  MoveL 8876 to (499.7, 501.14, 17.4) mm, rotated rx 0 ry 90 rz 0 deg; joints [-12.119, -28.128, 111.655, -16.143, -82.918, 51.024]
  Set speed (120.0 mm/s)
  MoveL 8877 to (499.36, 500.49, 17.4) mm, rotated rx 0 ry 90 rz 0 deg; joints [-12.066, -28.137, 111.711, -16.087, -82.962, 51.005]
  Set speed (15.0 mm/s)
  Call Extruder(0.050)
  MoveL 8878 to (500.58, 499.27, 17.4) mm, rotated rx 0 ry 90 rz 0 deg; joints [-11.93, -28.118, 111.596, -15.954, -82.865, 51.017]
  Set speed (120.0 mm/s)
  MoveL 8879 to (500.25, 498.61, 17.4) mm, rotated rx 0 ry 90 rz 0 deg; joints [-11.876, -28.127, 111.653, -15.898, -82.909, 50.998]
  Set speed (15.0 mm/s)
  MoveL 8880 to (499.03, 499.83, 17.4) mm, rotated rx 0 ry 90 rz 0 deg; joints [-12.012, -28.145, 111.768, -16.032, -83.006, 50.986]
  Set speed (120.0 mm/s)
  MoveL 8881 to (498.69, 499.17, 17.4) mm, rotated rx 0 ry 90 rz 0 deg; joints [-11.958, -28.154, 111.824, -15.976, -83.05, 50.967]
  Set speed (15.0 mm/s)
  Call Extruder(0.050)
  MoveL 8882 to (499.91, 497.96, 17.4) mm, rotated rx 0 ry 90 rz 0 deg; joints [-11.823, -28.136, 111.709, -15.843, -82.953, 50.979]
  Set speed (120.0 mm/s)
  MoveL 8883 to (499.58, 497.3, 17.4) mm, rotated rx 0 ry 90 rz 0 deg; joints [-11.769, -28.145, 111.766, -15.787, -82.997, 50.96]
  Set speed (15.0 mm/s)
  MoveL 8884 to (498.36, 498.52, 17.4) mm, rotated rx 0 ry 90 rz 0 deg; joints [-11.905, -28.163, 111.881, -15.92, -83.094, 50.948]
  Set speed (120.0 mm/s)
  MoveL 8885 to (498.02, 497.86, 17.4) mm, rotated rx 0 ry 90 rz 0 deg; joints [-11.851, -28.172, 111.937, -15.864, -83.138, 50.929]
  Set speed (15.0 mm/s)
  Call Extruder(0.050)
  MoveL 8886 to (499.24, 496.65, 17.4) mm, rotated rx 0 ry 90 rz 0 deg; joints [-11.715, -28.154, 111.822, -15.731, -83.041, 50.942]
  Set speed (120.0 mm/s)
  MoveL 8887 to (498.91, 495.99, 17.4) mm, rotated rx 0 ry 90 rz 0 deg; joints [-11.662, -28.163, 111.878, -15.676, -83.085, 50.923]
  Set speed (15.0 mm/s)
  Call Extruder(0.050)
  MoveL 8888 to (497.69, 497.21, 17.4) mm, rotated rx 0 ry 90 rz 0 deg; joints [-11.797, -28.181, 111.993, -15.809, -83.183, 50.911]
  Set speed (120.0 mm/s)
  MoveL 8889 to (497.36, 496.55, 17.4) mm, rotated rx 0 ry 90 rz 0 deg; joints [-11.743, -28.189, 112.049, -15.753, -83.227, 50.892]
  Set speed (15.0 mm/s)
  Call Extruder(0.107)
  MoveL 8890 to (499.95, 493.96, 17.4) mm, rotated rx 0 ry 90 rz 0 deg; joints [-11.455, -28.151, 111.804, -15.47, -83.018, 50.918]
  Set speed (120.0 mm/s)
  MoveL 8891 to (498.96, 493.96, 17.4) mm, rotated rx 0 ry 90 rz 0 deg; joints [-11.474, -28.17, 111.922, -15.485, -83.115, 50.893]
  Set speed (15.0 mm/s)
  Call Extruder(0.080)
  MoveL 8892 to (497.02, 495.9, 17.4) mm, rotated rx 0 ry 90 rz 0 deg; joints [-11.689, -28.198, 112.105, -15.697, -83.271, 50.874]
  Set speed (120.0 mm/s)
  MoveL 8893 to (496.69, 495.24, 17.4) mm, rotated rx 0 ry 90 rz 0 deg; joints [-11.635, -28.206, 112.161, -15.641, -83.315, 50.855]
  Set speed (15.0 mm/s)
  Call Extruder(0.053)
  MoveL 8894 to (497.97, 493.96, 17.4) mm, rotated rx 0 ry 90 rz 0 deg; joints [-11.492, -28.188, 112.04, -15.501, -83.212, 50.868]
  Set speed (120.0 mm/s)
  MoveL 8895 to (496.98, 493.96, 17.4) mm, rotated rx 0 ry 90 rz 0 deg; joints [-11.511, -28.206, 112.158, -15.516, -83.309, 50.843]
  Set speed (15.0 mm/s)
  Call Extruder(0.026)
  MoveL 8896 to (496.35, 494.59, 17.4) mm, rotated rx 0 ry 90 rz 0 deg; joints [-11.58, -28.215, 112.217, -15.585, -83.359, 50.837]
  Set speed (120.0 mm/s)
  MoveL 8897 to (499.33, 495.57, 17.4) mm, rotated rx 0 ry 90 rz 0 deg; joints [-11.614, -28.156, 111.838, -15.629, -83.051, 50.927]
  Set speed (15.0 mm/s)
  Call Extruder(0.066)
  MoveL 8898 to (500.94, 493.96, 17.4) mm, rotated rx 0 ry 90 rz 0 deg; joints [-11.437, -28.132, 111.685, -15.455, -82.922, 50.943]
  Set speed (120.0 mm/s)
  MoveL 8899 to (501.93, 493.96, 17.4) mm, rotated rx 0 ry 90 rz 0 deg; joints [-11.418, -28.114, 111.567, -15.44, -82.825, 50.968]
  Set speed (15.0 mm/s)
  MoveL 8900 to (500.32, 495.57, 17.4) mm, rotated rx 0 ry 90 rz 0 deg; joints [-11.596, -28.138, 111.719, -15.614, -82.954, 50.952]
  Set speed (120.0 mm/s)
  MoveL 8901 to (501.31, 495.57, 17.4) mm, rotated rx 0 ry 90 rz 0 deg; joints [-11.577, -28.119, 111.601, -15.598, -82.858, 50.977]
  Set speed (15.0 mm/s)
  MoveL 8902 to (502.92, 493.96, 17.4) mm, rotated rx 0 ry 90 rz 0 deg; joints [-11.4, -28.095, 111.448, -15.425, -82.728, 50.992]
  Set speed (120.0 mm/s)
  MoveL 8903 to (503.91, 493.96, 17.4) mm, rotated rx 0 ry 90 rz 0 deg; joints [-11.382, -28.076, 111.329, -15.41, -82.632, 51.017]
  Set speed (15.0 mm/s)
  MoveL 8904 to (502.3, 495.57, 17.4) mm, rotated rx 0 ry 90 rz 0 deg; joints [-11.558, -28.1, 111.483, -15.583, -82.761, 51.002]
  Set speed (120.0 mm/s)
  MoveL 8905 to (503.29, 495.56, 17.4) mm, rotated rx 0 ry 90 rz 0 deg; joints [-11.54, -28.081, 111.364, -15.568, -82.665, 51.027]
  Set speed (15.0 mm/s)
  Call Extruder(0.035)
  MoveL 8906 to (504.15, 494.7, 17.4) mm, rotated rx 0 ry 90 rz 0 deg; joints [-11.445, -28.068, 111.281, -15.475, -82.595, 51.035]
  Set speed (120.0 mm/s)
  MoveL 8907 to (502.26, 502.54, 17.4) mm, rotated rx 0 ry 90 rz 0 deg; joints [-12.196, -28.073, 111.312, -16.231, -82.644, 51.114]
  Set speed (15.0 mm/s)
  Call Extruder(0.050)
  MoveL 8908 to (501.03, 503.76, 17.4) mm, rotated rx 0 ry 90 rz 0 deg; joints [-12.332, -28.091, 111.427, -16.364, -82.741, 51.102]
  MoveL 8909 to (500.91, 503.89, 17.4) mm, rotated rx 0 ry 90 rz 0 deg; joints [-12.346, -28.093, 111.438, -16.378, -82.751, 51.101]
  Set speed (120.0 mm/s)
  MoveL 8910 to (490.68, 490.68, 17.4) mm, rotated rx 0 ry 90 rz 0 deg; joints [-11.324, -28.329, 112.985, -15.308, -83.983, 50.637]
  Set speed (1000.0 mm/s)
  MoveL 8911 to (490.68, 490.68, 17.5) mm, rotated rx 0 ry 90 rz 0 deg; joints [-11.324, -28.339, 112.99, -15.308, -83.977, 50.638]
  Set speed (30.0 mm/s)
  Call Extruder(0.287)
  MoveL 8912 to (497.65, 497.65, 17.5) mm, rotated rx 0 ry 90 rz 0 deg; joints [-11.838, -28.19, 111.992, -15.851, -83.173, 50.918]
  MoveL 8913 to (497.78, 497.78, 17.5) mm, rotated rx 0 ry 90 rz 0 deg; joints [-11.847, -28.187, 111.974, -15.86, -83.159, 50.923]
  Set speed (120.0 mm/s)
  MoveL 8914 to (499.24, 500.76, 17.5) mm, rotated rx 0 ry 90 rz 0 deg; joints [-12.093, -28.148, 111.724, -16.115, -82.964, 51.008]
  Set speed (30.0 mm/s)
  Call Extruder(0.352)
  MoveL 8915 to (490.68, 509.32, 17.5) mm, rotated rx 0 ry 90 rz 0 deg; joints [-13.056, -28.269, 112.514, -17.061, -83.634, 50.914]
  MoveL 8916 to (490.56, 509.44, 17.5) mm, rotated rx 0 ry 90 rz 0 deg; joints [-13.07, -28.271, 112.525, -17.075, -83.643, 50.913]
  Set speed (120.0 mm/s)
  MoveL 8917 to (496.13, 506.03, 17.5) mm, rotated rx 0 ry 90 rz 0 deg; joints [-12.639, -28.185, 111.957, -16.657, -83.169, 51.01]
  Set speed (30.0 mm/s)
  Call Extruder(0.224)
  MoveL 8918 to (490.68, 500.58, 17.5) mm, rotated rx 0 ry 90 rz 0 deg; joints [-12.247, -28.304, 112.746, -16.241, -83.8, 50.78]
  Set speed (120.0 mm/s)
  MoveL 8919 to (490.68, 499.42, 17.5) mm, rotated rx 0 ry 90 rz 0 deg; joints [-12.139, -28.308, 112.775, -16.132, -83.821, 50.763]
  Set speed (30.0 mm/s)
  Call Extruder(0.215)
  MoveL 8920 to (495.89, 494.21, 17.5) mm, rotated rx 0 ry 90 rz 0 deg; joints [-11.554, -28.235, 112.286, -15.557, -83.405, 50.821]
  Set speed (120.0 mm/s)
  MoveL 8921 to (496.37, 493.73, 17.5) mm, rotated rx 0 ry 90 rz 0 deg; joints [-11.5, -28.228, 112.241, -15.504, -83.367, 50.826]
  Set speed (30.0 mm/s)
  Call Extruder(0.125)
  MoveL 8922 to (499.42, 490.68, 17.5) mm, rotated rx 0 ry 90 rz 0 deg; joints [-11.163, -28.184, 111.95, -15.172, -83.12, 50.857]
  Set speed (120.0 mm/s)
  MoveL 8923 to (500.58, 490.68, 17.5) mm, rotated rx 0 ry 90 rz 0 deg; joints [-11.141, -28.162, 111.812, -15.154, -83.006, 50.885]
  Set speed (30.0 mm/s)
  MoveL 8924 to (503.63, 493.73, 17.5) mm, rotated rx 0 ry 90 rz 0 deg; joints [-11.366, -28.092, 111.374, -15.392, -82.658, 51.008]
  Set speed (120.0 mm/s)
  MoveL 8925 to (504.39, 494.49, 17.5) mm, rotated rx 0 ry 90 rz 0 deg; joints [-11.421, -28.075, 111.263, -15.451, -82.57, 51.039]
  Set speed (30.0 mm/s)
  Call Extruder(0.203)
  MoveL 8926 to (509.32, 499.42, 17.5) mm, rotated rx 0 ry 90 rz 0 deg; joints [-11.777, -27.956, 110.548, -15.832, -82.008, 51.244]
  Set speed (120.0 mm/s)
  MoveL 8927 to (509.32, 500.58, 17.5) mm, rotated rx 0 ry 90 rz 0 deg; joints [-11.882, -27.951, 110.519, -15.939, -81.988, 51.264]
  Set speed (30.0 mm/s)
  Call Extruder(0.212)
  MoveL 8928 to (504.16, 505.74, 17.5) mm, rotated rx 0 ry 90 rz 0 deg; joints [-12.449, -28.032, 111.006, -16.495, -82.397, 51.219]
  Set speed (120.0 mm/s)
  MoveL 8929 to (503.3, 506.6, 17.5) mm, rotated rx 0 ry 90 rz 0 deg; joints [-12.544, -28.046, 111.086, -16.589, -82.465, 51.211]
  Set speed (30.0 mm/s)
  Call Extruder(0.112)
  MoveL 8930 to (500.58, 509.32, 17.5) mm, rotated rx 0 ry 90 rz 0 deg; joints [-12.847, -28.087, 111.338, -16.886, -82.677, 51.184]
  Set speed (120.0 mm/s)
  MoveL 8931 to (499.42, 509.32, 17.5) mm, rotated rx 0 ry 90 rz 0 deg; joints [-12.872, -28.109, 111.476, -16.906, -82.789, 51.153]
  Set speed (30.0 mm/s)
  Call Extruder(0.112)
  MoveL 8932 to (496.7, 506.6, 17.5) mm, rotated rx 0 ry 90 rz 0 deg; joints [-12.679, -28.172, 111.874, -16.701, -83.103, 51.035]
  MoveL 8933 to (496.57, 506.47, 17.5) mm, rotated rx 0 ry 90 rz 0 deg; joints [-12.67, -28.175, 111.892, -16.691, -83.118, 51.029]
  Set speed (120.0 mm/s)
  MoveL 8934 to (502.51, 502.51, 17.5) mm, rotated rx 0 ry 90 rz 0 deg; joints [-12.188, -28.079, 111.289, -16.224, -82.615, 51.121]
  Set speed (30.0 mm/s)
  Call Extruder(0.280)
  MoveL 8935 to (509.32, 509.32, 17.5) mm, rotated rx 0 ry 90 rz 0 deg; joints [-12.669, -27.912, 110.29, -16.74, -81.835, 51.418]
  MoveL 8936 to (509.44, 509.44, 17.5) mm, rotated rx 0 ry 90 rz 0 deg; joints [-12.677, -27.908, 110.272, -16.75, -81.821, 51.423]
  Set speed (120.0 mm/s)
  MoveL 8937 to (500.81, 499.19, 17.5) mm, rotated rx 0 ry 90 rz 0 deg; joints [-11.919, -28.125, 111.576, -15.943, -82.839, 51.023]
  Set speed (30.0 mm/s)
  Call Extruder(0.140)
  MoveL 8938 to (504.2, 495.8, 17.5) mm, rotated rx 0 ry 90 rz 0 deg; joints [-11.544, -28.073, 111.255, -15.576, -82.567, 51.055]
  Set speed (120.0 mm/s)
  MoveL 8939 to (504.39, 495.61, 17.5) mm, rotated rx 0 ry 90 rz 0 deg; joints [-11.523, -28.07, 111.236, -15.555, -82.552, 51.057]
  Set speed (30.0 mm/s)
  Call Extruder(0.203)
  MoveL 8940 to (509.32, 490.68, 17.5) mm, rotated rx 0 ry 90 rz 0 deg; joints [-10.985, -27.992, 110.761, -15.026, -82.151, 51.098]
  MoveL 8941 to (509.44, 490.56, 17.5) mm, rotated rx 0 ry 90 rz 0 deg; joints [-10.972, -27.99, 110.749, -15.013, -82.141, 51.099]
  Set speed (120.0 mm/s)
  MoveL 8942 to (490.47, 509.53, 17.5) mm, rotated rx 0 ry 90 rz 0 deg; joints [-13.08, -28.272, 112.533, -17.085, -83.65, 50.912]
  Set speed (1000.0 mm/s)
  MoveL 8943 to (490.4, 509.6, 17.5) mm, rotated rx 0 ry 90 rz 0 deg; joints [-13.088, -28.273, 112.539, -17.093, -83.655, 50.911]
  Set speed (15.0 mm/s)
  Call Extruder(0.559)
  MoveL 8944 to (490.4, 490.4, 17.5) mm, rotated rx 0 ry 90 rz 0 deg; joints [-11.303, -28.345, 113.03, -15.286, -84.009, 50.628]
  MoveL 8945 to (509.6, 490.4, 17.5) mm, rotated rx 0 ry 90 rz 0 deg; joints [-10.955, -27.987, 110.733, -14.997, -82.128, 51.101]
  MoveL 8946 to (509.6, 509.6, 17.5) mm, rotated rx 0 ry 90 rz 0 deg; joints [-12.688, -27.904, 110.248, -16.761, -81.803, 51.43]
  MoveL 8947 to (490.4, 509.6, 17.5) mm, rotated rx 0 ry 90 rz 0 deg; joints [-13.088, -28.273, 112.539, -17.093, -83.655, 50.911]
  Set speed (120.0 mm/s)
  MoveL 8948 to (490.4, 509.2, 17.5) mm, rotated rx 0 ry 90 rz 0 deg; joints [-13.051, -28.275, 112.55, -17.055, -83.663, 50.905]
  Set speed (1000.0 mm/s)
  MoveL 8949 to (490.5, 509.2, 17.5) mm, rotated rx 0 ry 90 rz 0 deg; joints [-13.049, -28.273, 112.538, -17.054, -83.653, 50.908]
  Set speed (1000.0 mm/s)
  MoveL 8950 to (496.05, 506.68, 17.5) mm, rotated rx 0 ry 90 rz 0 deg; joints [-12.7, -28.184, 111.949, -16.719, -83.165, 51.018]
  Set speed (15.0 mm/s)
  Call Extruder(0.065)
  MoveL 8951 to (496.05, 504.44, 17.5) mm, rotated rx 0 ry 90 rz 0 deg; joints [-12.495, -28.193, 112.009, -16.511, -83.207, 50.983]
  Call Extruder(0.145)
  MoveL 8952 to (501.03, 504.44, 17.5) mm, rotated rx 0 ry 90 rz 0 deg; joints [-12.394, -28.099, 111.415, -16.428, -82.724, 51.115]
  Call Extruder(0.353)
  MoveL 8953 to (495.52, 493.65, 17.5) mm, rotated rx 0 ry 90 rz 0 deg; joints [-11.509, -28.244, 112.344, -15.51, -83.451, 50.803]
  Call Extruder(0.261)
  MoveL 8954 to (504.47, 493.65, 17.5) mm, rotated rx 0 ry 90 rz 0 deg; joints [-11.343, -28.076, 111.274, -15.372, -82.576, 51.027]
  Call Extruder(0.065)
  MoveL 8955 to (504.47, 495.88, 17.5) mm, rotated rx 0 ry 90 rz 0 deg; joints [-11.547, -28.068, 111.22, -15.579, -82.539, 51.063]
  Call Extruder(0.153)
  MoveL 8956 to (499.2, 495.88, 17.5) mm, rotated rx 0 ry 90 rz 0 deg; joints [-11.646, -28.168, 111.85, -15.661, -83.053, 50.93]
  Call Extruder(0.353)
  MoveL 8957 to (504.73, 506.68, 17.5) mm, rotated rx 0 ry 90 rz 0 deg; joints [-12.523, -28.017, 110.912, -16.573, -82.325, 51.25]
  Call Extruder(0.253)
  MoveL 8958 to (496.05, 506.68, 17.5) mm, rotated rx 0 ry 90 rz 0 deg; joints [-12.7, -28.184, 111.949, -16.719, -83.165, 51.018]
  Set speed (120.0 mm/s)
  MoveL 8959 to (496.46, 506.36, 17.5) mm, rotated rx 0 ry 90 rz 0 deg; joints [-12.662, -28.177, 111.908, -16.683, -83.131, 51.025]
  Set speed (15.0 mm/s)
  Call Extruder(0.004)
  MoveL 8960 to (496.36, 506.26, 17.5) mm, rotated rx 0 ry 90 rz 0 deg; joints [-12.655, -28.18, 111.923, -16.675, -83.142, 51.02]
  Set speed (120.0 mm/s)
  MoveL 8961 to (496.36, 505.27, 17.5) mm, rotated rx 0 ry 90 rz 0 deg; joints [-12.564, -28.184, 111.95, -16.583, -83.161, 51.004]
  Set speed (15.0 mm/s)
  Call Extruder(0.045)
  MoveL 8962 to (497.45, 506.36, 17.5) mm, rotated rx 0 ry 90 rz 0 deg; joints [-12.642, -28.159, 111.791, -16.666, -83.035, 51.051]
  Set speed (120.0 mm/s)
  MoveL 8963 to (498.44, 506.36, 17.5) mm, rotated rx 0 ry 90 rz 0 deg; joints [-12.622, -28.14, 111.673, -16.649, -82.939, 51.078]
  Set speed (15.0 mm/s)
  Call Extruder(0.066)
  MoveL 8964 to (496.84, 504.76, 17.5) mm, rotated rx 0 ry 90 rz 0 deg; joints [-12.508, -28.177, 111.906, -16.527, -83.124, 51.009]
  Set speed (120.0 mm/s)
  MoveL 8965 to (497.83, 504.76, 17.5) mm, rotated rx 0 ry 90 rz 0 deg; joints [-12.488, -28.158, 111.788, -16.51, -83.028, 51.035]
  Set speed (15.0 mm/s)
  MoveL 8966 to (499.43, 506.36, 17.5) mm, rotated rx 0 ry 90 rz 0 deg; joints [-12.602, -28.121, 111.555, -16.632, -82.843, 51.104]
  Set speed (120.0 mm/s)
  MoveL 8967 to (500.42, 506.36, 17.5) mm, rotated rx 0 ry 90 rz 0 deg; joints [-12.581, -28.103, 111.437, -16.615, -82.747, 51.13]
  Set speed (15.0 mm/s)
  MoveL 8968 to (498.82, 504.76, 17.5) mm, rotated rx 0 ry 90 rz 0 deg; joints [-12.468, -28.14, 111.67, -16.493, -82.932, 51.061]
  Set speed (120.0 mm/s)
  MoveL 8969 to (499.81, 504.76, 17.5) mm, rotated rx 0 ry 90 rz 0 deg; joints [-12.448, -28.121, 111.552, -16.477, -82.836, 51.088]
  Set speed (15.0 mm/s)
  MoveL 8970 to (501.41, 506.36, 17.5) mm, rotated rx 0 ry 90 rz 0 deg; joints [-12.561, -28.083, 111.318, -16.599, -82.652, 51.157]
  Set speed (120.0 mm/s)
  MoveL 8971 to (502.4, 506.36, 17.5) mm, rotated rx 0 ry 90 rz 0 deg; joints [-12.541, -28.064, 111.2, -16.582, -82.556, 51.183]
  Set speed (15.0 mm/s)
  MoveL 8972 to (500.8, 504.76, 17.5) mm, rotated rx 0 ry 90 rz 0 deg; joints [-12.428, -28.102, 111.434, -16.46, -82.74, 51.114]
  Set speed (120.0 mm/s)
  MoveL 8973 to (501.28, 504.25, 17.5) mm, rotated rx 0 ry 90 rz 0 deg; joints [-12.372, -28.095, 111.389, -16.406, -82.703, 51.118]
  Set speed (15.0 mm/s)
  Call Extruder(0.087)
  MoveL 8974 to (503.39, 506.36, 17.5) mm, rotated rx 0 ry 90 rz 0 deg; joints [-12.521, -28.045, 111.081, -16.566, -82.46, 51.209]
  Set speed (120.0 mm/s)
  MoveL 8975 to (504.04, 506.02, 17.5) mm, rotated rx 0 ry 90 rz 0 deg; joints [-12.477, -28.034, 111.013, -16.523, -82.404, 51.22]
  Set speed (15.0 mm/s)
  Call Extruder(0.156)
  MoveL 8976 to (500.25, 502.23, 17.5) mm, rotated rx 0 ry 90 rz 0 deg; joints [-12.208, -28.123, 111.565, -16.235, -82.839, 51.058]
  MoveL 8977 to (500.13, 502.11, 17.5) mm, rotated rx 0 ry 90 rz 0 deg; joints [-12.199, -28.126, 111.583, -16.226, -82.853, 51.053]
  Set speed (120.0 mm/s)
  MoveL 8978 to (501.96, 501.96, 17.5) mm, rotated rx 0 ry 90 rz 0 deg; joints [-12.15, -28.091, 111.367, -16.182, -82.678, 51.098]
  Set speed (15.0 mm/s)
  Call Extruder(0.155)
  MoveL 8979 to (498.19, 498.19, 17.5) mm, rotated rx 0 ry 90 rz 0 deg; joints [-11.878, -28.178, 111.914, -15.892, -83.111, 50.94]
  MoveL 8980 to (498.07, 498.07, 17.5) mm, rotated rx 0 ry 90 rz 0 deg; joints [-11.869, -28.181, 111.932, -15.883, -83.125, 50.935]
  Set speed (120.0 mm/s)
  MoveL 8981 to (499.89, 497.91, 17.5) mm, rotated rx 0 ry 90 rz 0 deg; joints [-11.819, -28.147, 111.718, -15.839, -82.951, 50.979]
  Set speed (15.0 mm/s)
  Call Extruder(0.155)
  MoveL 8982 to (496.13, 494.15, 17.5) mm, rotated rx 0 ry 90 rz 0 deg; joints [-11.544, -28.231, 112.26, -15.548, -83.383, 50.826]
  Set speed (120.0 mm/s)
  MoveL 8983 to (496.93, 493.96, 17.5) mm, rotated rx 0 ry 90 rz 0 deg; joints [-11.512, -28.217, 112.168, -15.517, -83.308, 50.844]
  Set speed (15.0 mm/s)
  Call Extruder(0.079)
  MoveL 8984 to (498.85, 495.88, 17.5) mm, rotated rx 0 ry 90 rz 0 deg; joints [-11.652, -28.175, 111.893, -15.666, -83.087, 50.921]
  Set speed (120.0 mm/s)
  MoveL 8985 to (499.52, 495.56, 17.5) mm, rotated rx 0 ry 90 rz 0 deg; joints [-11.611, -28.163, 111.82, -15.626, -83.027, 50.934]
  Set speed (15.0 mm/s)
  Call Extruder(0.066)
  MoveL 8986 to (497.92, 493.96, 17.5) mm, rotated rx 0 ry 90 rz 0 deg; joints [-11.493, -28.199, 112.051, -15.502, -83.211, 50.869]
  Set speed (120.0 mm/s)
  MoveL 8987 to (498.91, 493.96, 17.5) mm, rotated rx 0 ry 90 rz 0 deg; joints [-11.475, -28.181, 111.932, -15.486, -83.114, 50.894]
  Set speed (15.0 mm/s)
  MoveL 8988 to (500.51, 495.57, 17.5) mm, rotated rx 0 ry 90 rz 0 deg; joints [-11.592, -28.145, 111.702, -15.611, -82.93, 50.959]
  Set speed (120.0 mm/s)
  MoveL 8989 to (501.5, 495.56, 17.5) mm, rotated rx 0 ry 90 rz 0 deg; joints [-11.573, -28.126, 111.583, -15.595, -82.834, 50.984]
  Set speed (15.0 mm/s)
  MoveL 8990 to (499.9, 493.96, 17.5) mm, rotated rx 0 ry 90 rz 0 deg; joints [-11.456, -28.162, 111.814, -15.471, -83.018, 50.918]
  Set speed (120.0 mm/s)
  MoveL 8991 to (500.89, 493.96, 17.5) mm, rotated rx 0 ry 90 rz 0 deg; joints [-11.438, -28.144, 111.696, -15.456, -82.921, 50.943]
  Set speed (15.0 mm/s)
  MoveL 8992 to (502.49, 495.56, 17.5) mm, rotated rx 0 ry 90 rz 0 deg; joints [-11.555, -28.107, 111.465, -15.58, -82.737, 51.009]
  Set speed (120.0 mm/s)
  MoveL 8993 to (503.48, 495.56, 17.5) mm, rotated rx 0 ry 90 rz 0 deg; joints [-11.536, -28.088, 111.346, -15.565, -82.641, 51.033]
  Set speed (15.0 mm/s)
  MoveL 8994 to (501.88, 493.96, 17.5) mm, rotated rx 0 ry 90 rz 0 deg; joints [-11.419, -28.125, 111.577, -15.44, -82.824, 50.968]
  Set speed (120.0 mm/s)
  MoveL 8995 to (502.87, 493.96, 17.5) mm, rotated rx 0 ry 90 rz 0 deg; joints [-11.401, -28.106, 111.459, -15.425, -82.727, 50.993]
  Set speed (15.0 mm/s)
  Call Extruder(0.053)
  MoveL 8996 to (504.16, 495.25, 17.5) mm, rotated rx 0 ry 90 rz 0 deg; joints [-11.495, -28.076, 111.273, -15.525, -82.581, 51.045]
  Set speed (120.0 mm/s)
  MoveL 8997 to (504.16, 494.26, 17.5) mm, rotated rx 0 ry 90 rz 0 deg; joints [-11.404, -28.08, 111.297, -15.433, -82.597, 51.029]
  Set speed (15.0 mm/s)
  Call Extruder(0.012)
  MoveL 8998 to (503.86, 493.96, 17.5) mm, rotated rx 0 ry 90 rz 0 deg; joints [-11.383, -28.087, 111.34, -15.41, -82.631, 51.017]
  Set speed (120.0 mm/s)
  MoveL 8999 to (500.93, 499.94, 17.5) mm, rotated rx 0 ry 90 rz 0 deg; joints [-11.985, -28.12, 111.543, -16.011, -82.814, 51.038]
  Set speed (15.0 mm/s)
  Call Extruder(0.155)
  MoveL 9000 to (497.16, 496.17, 17.5) mm, rotated rx 0 ry 90 rz 0 deg; joints [-11.711, -28.205, 112.087, -15.72, -83.247, 50.883]
  MoveL 9001 to (497.04, 496.05, 17.5) mm, rotated rx 0 ry 90 rz 0 deg; joints [-11.702, -28.208, 112.105, -15.711, -83.261, 50.878]
  Set speed (120.0 mm/s)
  MoveL 9002 to (499.22, 500.21, 17.5) mm, rotated rx 0 ry 90 rz 0 deg; joints [-12.043, -28.151, 111.74, -16.064, -82.975, 50.999]
  Set speed (15.0 mm/s)
  Call Extruder(0.156)
  MoveL 9003 to (503, 503.99, 17.5) mm, rotated rx 0 ry 90 rz 0 deg; joints [-12.314, -28.063, 111.19, -16.353, -82.541, 51.159]
  MoveL 9004 to (503.13, 504.12, 17.5) mm, rotated rx 0 ry 90 rz 0 deg; joints [-12.323, -28.06, 111.173, -16.363, -82.527, 51.164]
  Set speed (120.0 mm/s)
  MoveL 9005 to (490.68, 490.68, 17.5) mm, rotated rx 0 ry 90 rz 0 deg; joints [-11.324, -28.339, 112.99, -15.308, -83.977, 50.638]
  Set speed (1000.0 mm/s)
  MoveL 9006 to (490.68, 490.68, 17.6) mm, rotated rx 0 ry 90 rz 0 deg; joints [-11.324, -28.35, 112.995, -15.308, -83.972, 50.64]
  Set speed (30.0 mm/s)
  Call Extruder(0.287)
  MoveL 9007 to (497.65, 497.65, 17.6) mm, rotated rx 0 ry 90 rz 0 deg; joints [-11.838, -28.201, 111.997, -15.851, -83.168, 50.92]
  MoveL 9008 to (497.78, 497.78, 17.6) mm, rotated rx 0 ry 90 rz 0 deg; joints [-11.847, -28.198, 111.979, -15.861, -83.154, 50.925]
  Set speed (120.0 mm/s)
  MoveL 9009 to (499.24, 500.76, 17.6) mm, rotated rx 0 ry 90 rz 0 deg; joints [-12.093, -28.159, 111.729, -16.115, -82.959, 51.009]
  Set speed (30.0 mm/s)
  Call Extruder(0.352)
  MoveL 9010 to (490.68, 509.32, 17.6) mm, rotated rx 0 ry 90 rz 0 deg; joints [-13.056, -28.28, 112.519, -17.062, -83.628, 50.916]
  MoveL 9011 to (490.56, 509.44, 17.6) mm, rotated rx 0 ry 90 rz 0 deg; joints [-13.07, -28.282, 112.53, -17.075, -83.638, 50.915]
  Set speed (120.0 mm/s)
  MoveL 9012 to (496.13, 506.03, 17.6) mm, rotated rx 0 ry 90 rz 0 deg; joints [-12.639, -28.195, 111.962, -16.658, -83.164, 51.012]
  Set speed (30.0 mm/s)
  Call Extruder(0.224)
  MoveL 9013 to (490.68, 500.58, 17.6) mm, rotated rx 0 ry 90 rz 0 deg; joints [-12.247, -28.314, 112.751, -16.242, -83.795, 50.782]
  Set speed (120.0 mm/s)
  MoveL 9014 to (490.68, 499.42, 17.6) mm, rotated rx 0 ry 90 rz 0 deg; joints [-12.139, -28.319, 112.78, -16.132, -83.816, 50.765]
  Set speed (30.0 mm/s)
  Call Extruder(0.215)
  MoveL 9015 to (495.89, 494.21, 17.6) mm, rotated rx 0 ry 90 rz 0 deg; joints [-11.554, -28.246, 112.291, -15.557, -83.4, 50.822]
  Set speed (120.0 mm/s)
  MoveL 9016 to (496.37, 493.73, 17.6) mm, rotated rx 0 ry 90 rz 0 deg; joints [-11.5, -28.239, 112.246, -15.504, -83.361, 50.827]
  Set speed (30.0 mm/s)
  Call Extruder(0.125)
  MoveL 9017 to (499.42, 490.68, 17.6) mm, rotated rx 0 ry 90 rz 0 deg; joints [-11.163, -28.194, 111.955, -15.172, -83.114, 50.858]
  Set speed (120.0 mm/s)
  MoveL 9018 to (500.58, 490.68, 17.6) mm, rotated rx 0 ry 90 rz 0 deg; joints [-11.141, -28.173, 111.817, -15.154, -83.001, 50.887]
  Set speed (30.0 mm/s)
  MoveL 9019 to (503.63, 493.73, 17.6) mm, rotated rx 0 ry 90 rz 0 deg; joints [-11.366, -28.103, 111.379, -15.392, -82.652, 51.009]
  Set speed (120.0 mm/s)
  MoveL 9020 to (504.39, 494.49, 17.6) mm, rotated rx 0 ry 90 rz 0 deg; joints [-11.421, -28.085, 111.268, -15.452, -82.565, 51.04]
  Set speed (30.0 mm/s)
  Call Extruder(0.203)
  MoveL 9021 to (509.32, 499.42, 17.6) mm, rotated rx 0 ry 90 rz 0 deg; joints [-11.777, -27.966, 110.553, -15.832, -82.003, 51.245]
  Set speed (120.0 mm/s)
  MoveL 9022 to (509.32, 500.58, 17.6) mm, rotated rx 0 ry 90 rz 0 deg; joints [-11.882, -27.961, 110.524, -15.939, -81.983, 51.265]
  Set speed (30.0 mm/s)
  Call Extruder(0.212)
  MoveL 9023 to (504.16, 505.74, 17.6) mm, rotated rx 0 ry 90 rz 0 deg; joints [-12.449, -28.043, 111.011, -16.496, -82.392, 51.22]
  Set speed (120.0 mm/s)
  MoveL 9024 to (503.3, 506.6, 17.6) mm, rotated rx 0 ry 90 rz 0 deg; joints [-12.544, -28.056, 111.091, -16.589, -82.46, 51.212]
  Set speed (30.0 mm/s)
  Call Extruder(0.112)
  MoveL 9025 to (500.58, 509.32, 17.6) mm, rotated rx 0 ry 90 rz 0 deg; joints [-12.847, -28.097, 111.343, -16.887, -82.672, 51.186]
  Set speed (120.0 mm/s)
  MoveL 9026 to (499.42, 509.32, 17.6) mm, rotated rx 0 ry 90 rz 0 deg; joints [-12.872, -28.12, 111.482, -16.906, -82.784, 51.155]
  Set speed (30.0 mm/s)
  Call Extruder(0.112)
  MoveL 9027 to (496.7, 506.6, 17.6) mm, rotated rx 0 ry 90 rz 0 deg; joints [-12.679, -28.182, 111.879, -16.701, -83.098, 51.036]
  MoveL 9028 to (496.57, 506.47, 17.6) mm, rotated rx 0 ry 90 rz 0 deg; joints [-12.67, -28.185, 111.897, -16.691, -83.112, 51.031]
  Set speed (120.0 mm/s)
  MoveL 9029 to (502.51, 502.51, 17.6) mm, rotated rx 0 ry 90 rz 0 deg; joints [-12.188, -28.089, 111.294, -16.224, -82.61, 51.123]
  Set speed (30.0 mm/s)
  Call Extruder(0.280)
  MoveL 9030 to (509.32, 509.32, 17.6) mm, rotated rx 0 ry 90 rz 0 deg; joints [-12.669, -27.922, 110.295, -16.741, -81.83, 51.419]
  MoveL 9031 to (509.44, 509.44, 17.6) mm, rotated rx 0 ry 90 rz 0 deg; joints [-12.677, -27.919, 110.277, -16.75, -81.816, 51.425]
  Set speed (120.0 mm/s)
  MoveL 9032 to (500.81, 499.19, 17.6) mm, rotated rx 0 ry 90 rz 0 deg; joints [-11.919, -28.135, 111.581, -15.944, -82.834, 51.025]
  Set speed (30.0 mm/s)
  Call Extruder(0.140)
  MoveL 9033 to (504.2, 495.8, 17.6) mm, rotated rx 0 ry 90 rz 0 deg; joints [-11.544, -28.084, 111.26, -15.576, -82.562, 51.057]
  Set speed (120.0 mm/s)
  MoveL 9034 to (504.39, 495.61, 17.6) mm, rotated rx 0 ry 90 rz 0 deg; joints [-11.523, -28.081, 111.241, -15.555, -82.546, 51.058]
  Set speed (30.0 mm/s)
  Call Extruder(0.203)
  MoveL 9035 to (509.32, 490.68, 17.6) mm, rotated rx 0 ry 90 rz 0 deg; joints [-10.985, -28.002, 110.766, -15.027, -82.146, 51.1]
  MoveL 9036 to (509.44, 490.56, 17.6) mm, rotated rx 0 ry 90 rz 0 deg; joints [-10.972, -28, 110.754, -15.014, -82.136, 51.101]
  Set speed (120.0 mm/s)
  MoveL 9037 to (490.47, 509.53, 17.6) mm, rotated rx 0 ry 90 rz 0 deg; joints [-13.08, -28.283, 112.538, -17.085, -83.644, 50.914]
  Set speed (1000.0 mm/s)
  MoveL 9038 to (490.4, 509.6, 17.6) mm, rotated rx 0 ry 90 rz 0 deg; joints [-13.088, -28.284, 112.544, -17.093, -83.65, 50.913]
  Set speed (15.0 mm/s)
  Call Extruder(0.559)
  MoveL 9039 to (490.4, 490.4, 17.6) mm, rotated rx 0 ry 90 rz 0 deg; joints [-11.303, -28.356, 113.035, -15.286, -84.004, 50.629]
  MoveL 9040 to (509.6, 490.4, 17.6) mm, rotated rx 0 ry 90 rz 0 deg; joints [-10.955, -27.998, 110.738, -14.997, -82.123, 51.102]
  MoveL 9041 to (509.6, 509.6, 17.6) mm, rotated rx 0 ry 90 rz 0 deg; joints [-12.688, -27.915, 110.253, -16.762, -81.798, 51.432]
  MoveL 9042 to (490.4, 509.6, 17.6) mm, rotated rx 0 ry 90 rz 0 deg; joints [-13.088, -28.284, 112.544, -17.093, -83.65, 50.913]
  Set speed (120.0 mm/s)
  MoveL 9043 to (490.4, 509.2, 17.6) mm, rotated rx 0 ry 90 rz 0 deg; joints [-13.051, -28.286, 112.555, -17.056, -83.658, 50.906]
  Set speed (1000.0 mm/s)
  MoveL 9044 to (490.5, 509.2, 17.6) mm, rotated rx 0 ry 90 rz 0 deg; joints [-13.049, -28.284, 112.543, -17.054, -83.648, 50.909]
  Set speed (1000.0 mm/s)
  MoveL 9045 to (496.05, 506.68, 17.6) mm, rotated rx 0 ry 90 rz 0 deg; joints [-12.7, -28.194, 111.954, -16.72, -83.16, 51.02]
  Set speed (15.0 mm/s)
  Call Extruder(0.065)
  MoveL 9046 to (496.05, 504.44, 17.6) mm, rotated rx 0 ry 90 rz 0 deg; joints [-12.495, -28.203, 112.014, -16.512, -83.201, 50.984]
  Call Extruder(0.145)
  MoveL 9047 to (501.03, 504.45, 17.6) mm, rotated rx 0 ry 90 rz 0 deg; joints [-12.394, -28.11, 111.42, -16.428, -82.719, 51.116]
  Call Extruder(0.353)
  MoveL 9048 to (495.52, 493.65, 17.6) mm, rotated rx 0 ry 90 rz 0 deg; joints [-11.509, -28.255, 112.349, -15.51, -83.446, 50.805]
  Call Extruder(0.261)
  MoveL 9049 to (504.47, 493.65, 17.6) mm, rotated rx 0 ry 90 rz 0 deg; joints [-11.343, -28.087, 111.279, -15.372, -82.571, 51.029]
  Call Extruder(0.065)
  MoveL 9050 to (504.47, 495.88, 17.6) mm, rotated rx 0 ry 90 rz 0 deg; joints [-11.547, -28.078, 111.225, -15.579, -82.534, 51.065]
  Call Extruder(0.153)
  MoveL 9051 to (499.2, 495.88, 17.6) mm, rotated rx 0 ry 90 rz 0 deg; joints [-11.646, -28.179, 111.856, -15.661, -83.047, 50.932]
  Call Extruder(0.353)
  MoveL 9052 to (504.73, 506.68, 17.6) mm, rotated rx 0 ry 90 rz 0 deg; joints [-12.523, -28.027, 110.918, -16.573, -82.32, 51.251]
  Call Extruder(0.253)
  MoveL 9053 to (496.05, 506.68, 17.6) mm, rotated rx 0 ry 90 rz 0 deg; joints [-12.7, -28.194, 111.954, -16.72, -83.16, 51.02]
  Set speed (120.0 mm/s)
  MoveL 9054 to (503.93, 505.81, 17.6) mm, rotated rx 0 ry 90 rz 0 deg; joints [-12.461, -28.047, 111.036, -16.506, -82.413, 51.216]
  Set speed (15.0 mm/s)
  Call Extruder(0.023)
  MoveL 9055 to (503.39, 506.36, 17.6) mm, rotated rx 0 ry 90 rz 0 deg; joints [-12.521, -28.055, 111.087, -16.566, -82.456, 51.211]
  Set speed (120.0 mm/s)
  MoveL 9056 to (502.4, 506.36, 17.6) mm, rotated rx 0 ry 90 rz 0 deg; joints [-12.541, -28.075, 111.206, -16.582, -82.551, 51.184]
  Set speed (15.0 mm/s)
  Call Extruder(0.049)
  MoveL 9057 to (503.6, 505.16, 17.6) mm, rotated rx 0 ry 90 rz 0 deg; joints [-12.408, -28.057, 111.093, -16.451, -82.457, 51.196]
  Set speed (120.0 mm/s)
  MoveL 9058 to (503.26, 504.5, 17.6) mm, rotated rx 0 ry 90 rz 0 deg; joints [-12.355, -28.066, 111.151, -16.396, -82.501, 51.176]
  Set speed (15.0 mm/s)
  Call Extruder(0.076)
  MoveL 9059 to (501.41, 506.36, 17.6) mm, rotated rx 0 ry 90 rz 0 deg; joints [-12.561, -28.094, 111.324, -16.599, -82.647, 51.158]
  Set speed (120.0 mm/s)
  MoveL 9060 to (500.42, 506.36, 17.6) mm, rotated rx 0 ry 90 rz 0 deg; joints [-12.581, -28.113, 111.442, -16.615, -82.743, 51.132]
  Set speed (15.0 mm/s)
  Call Extruder(0.103)
  MoveL 9061 to (502.93, 503.85, 17.6) mm, rotated rx 0 ry 90 rz 0 deg; joints [-12.302, -28.075, 111.208, -16.341, -82.545, 51.156]
  Set speed (120.0 mm/s)
  MoveL 9062 to (502.59, 503.19, 17.6) mm, rotated rx 0 ry 90 rz 0 deg; joints [-12.249, -28.085, 111.265, -16.286, -82.589, 51.136]
  Set speed (15.0 mm/s)
  Call Extruder(0.050)
  MoveL 9063 to (501.37, 504.42, 17.6) mm, rotated rx 0 ry 90 rz 0 deg; joints [-12.385, -28.103, 111.38, -16.42, -82.686, 51.125]
  Set speed (120.0 mm/s)
  MoveL 9064 to (501.03, 504.76, 17.6) mm, rotated rx 0 ry 90 rz 0 deg; joints [-12.423, -28.108, 111.412, -16.457, -82.713, 51.121]
  Set speed (15.0 mm/s)
  Call Extruder(0.066)
  MoveL 9065 to (499.43, 506.36, 17.6) mm, rotated rx 0 ry 90 rz 0 deg; joints [-12.602, -28.132, 111.56, -16.632, -82.839, 51.105]
  Set speed (120.0 mm/s)
  MoveL 9066 to (498.44, 506.36, 17.6) mm, rotated rx 0 ry 90 rz 0 deg; joints [-12.622, -28.151, 111.678, -16.649, -82.934, 51.079]
  Set speed (15.0 mm/s)
  MoveL 9067 to (500.04, 504.76, 17.6) mm, rotated rx 0 ry 90 rz 0 deg; joints [-12.443, -28.127, 111.53, -16.473, -82.809, 51.095]
  Set speed (120.0 mm/s)
  MoveL 9068 to (499.05, 504.76, 17.6) mm, rotated rx 0 ry 90 rz 0 deg; joints [-12.463, -28.146, 111.648, -16.49, -82.905, 51.069]
  Set speed (15.0 mm/s)
  MoveL 9069 to (497.45, 506.36, 17.6) mm, rotated rx 0 ry 90 rz 0 deg; joints [-12.642, -28.169, 111.796, -16.666, -83.03, 51.053]
  Set speed (120.0 mm/s)
  MoveL 9070 to (496.46, 506.36, 17.6) mm, rotated rx 0 ry 90 rz 0 deg; joints [-12.663, -28.188, 111.914, -16.683, -83.126, 51.026]
  Set speed (15.0 mm/s)
  MoveL 9071 to (498.06, 504.76, 17.6) mm, rotated rx 0 ry 90 rz 0 deg; joints [-12.483, -28.165, 111.766, -16.506, -83, 51.043]
  Set speed (120.0 mm/s)
  MoveL 9072 to (497.07, 504.76, 17.6) mm, rotated rx 0 ry 90 rz 0 deg; joints [-12.503, -28.183, 111.884, -16.523, -83.096, 51.016]
  Set speed (15.0 mm/s)
  Call Extruder(0.029)
  MoveL 9073 to (496.36, 505.47, 17.6) mm, rotated rx 0 ry 90 rz 0 deg; joints [-12.583, -28.193, 111.949, -16.601, -83.152, 51.009]
  Set speed (120.0 mm/s)
  MoveL 9074 to (500.7, 503.11, 17.6) mm, rotated rx 0 ry 90 rz 0 deg; joints [-12.279, -28.122, 111.494, -16.309, -82.774, 51.086]
  Set speed (15.0 mm/s)
  Call Extruder(0.050)
  MoveL 9075 to (501.92, 501.89, 17.6) mm, rotated rx 0 ry 90 rz 0 deg; joints [-12.143, -28.103, 111.379, -16.176, -82.678, 51.097]
  Set speed (120.0 mm/s)
  MoveL 9076 to (501.59, 501.23, 17.6) mm, rotated rx 0 ry 90 rz 0 deg; joints [-12.09, -28.112, 111.436, -16.121, -82.722, 51.078]
  Set speed (15.0 mm/s)
  MoveL 9077 to (500.36, 502.45, 17.6) mm, rotated rx 0 ry 90 rz 0 deg; joints [-12.226, -28.131, 111.551, -16.254, -82.819, 51.066]
  Set speed (120.0 mm/s)
  MoveL 9078 to (500.03, 501.8, 17.6) mm, rotated rx 0 ry 90 rz 0 deg; joints [-12.172, -28.14, 111.608, -16.198, -82.863, 51.047]
  Set speed (15.0 mm/s)
  Call Extruder(0.050)
  MoveL 9079 to (501.25, 500.58, 17.6) mm, rotated rx 0 ry 90 rz 0 deg; joints [-12.037, -28.121, 111.493, -16.065, -82.766, 51.059]
  Set speed (120.0 mm/s)
  MoveL 9080 to (500.92, 499.92, 17.6) mm, rotated rx 0 ry 90 rz 0 deg; joints [-11.983, -28.13, 111.55, -16.01, -82.81, 51.039]
  Set speed (15.0 mm/s)
  Call Extruder(0.050)
  MoveL 9081 to (499.7, 501.14, 17.6) mm, rotated rx 0 ry 90 rz 0 deg; joints [-12.119, -28.149, 111.665, -16.143, -82.907, 51.027]
  Set speed (120.0 mm/s)
  MoveL 9082 to (499.36, 500.49, 17.6) mm, rotated rx 0 ry 90 rz 0 deg; joints [-12.066, -28.158, 111.721, -16.088, -82.951, 51.008]
  Set speed (15.0 mm/s)
  Call Extruder(0.050)
  MoveL 9083 to (500.58, 499.27, 17.6) mm, rotated rx 0 ry 90 rz 0 deg; joints [-11.93, -28.14, 111.607, -15.954, -82.854, 51.02]
  Set speed (120.0 mm/s)
  MoveL 9084 to (500.25, 498.61, 17.6) mm, rotated rx 0 ry 90 rz 0 deg; joints [-11.876, -28.148, 111.663, -15.899, -82.898, 51.001]
  Set speed (15.0 mm/s)
  MoveL 9085 to (499.03, 499.83, 17.6) mm, rotated rx 0 ry 90 rz 0 deg; joints [-12.012, -28.167, 111.778, -16.032, -82.996, 50.989]
  Set speed (120.0 mm/s)
  MoveL 9086 to (498.69, 499.17, 17.6) mm, rotated rx 0 ry 90 rz 0 deg; joints [-11.958, -28.175, 111.834, -15.976, -83.04, 50.97]
  Set speed (15.0 mm/s)
  Call Extruder(0.050)
  MoveL 9087 to (499.91, 497.96, 17.6) mm, rotated rx 0 ry 90 rz 0 deg; joints [-11.823, -28.157, 111.72, -15.843, -82.942, 50.982]
  Set speed (120.0 mm/s)
  MoveL 9088 to (499.58, 497.3, 17.6) mm, rotated rx 0 ry 90 rz 0 deg; joints [-11.769, -28.166, 111.776, -15.787, -82.986, 50.963]
  Set speed (15.0 mm/s)
  MoveL 9089 to (498.36, 498.52, 17.6) mm, rotated rx 0 ry 90 rz 0 deg; joints [-11.905, -28.184, 111.891, -15.921, -83.084, 50.951]
  Set speed (120.0 mm/s)
  MoveL 9090 to (498.02, 497.86, 17.6) mm, rotated rx 0 ry 90 rz 0 deg; joints [-11.851, -28.193, 111.947, -15.865, -83.128, 50.932]
  Set speed (15.0 mm/s)
  Call Extruder(0.050)
  MoveL 9091 to (499.24, 496.65, 17.6) mm, rotated rx 0 ry 90 rz 0 deg; joints [-11.715, -28.175, 111.832, -15.732, -83.03, 50.945]
  Set speed (120.0 mm/s)
  MoveL 9092 to (498.91, 495.99, 17.6) mm, rotated rx 0 ry 90 rz 0 deg; joints [-11.662, -28.184, 111.888, -15.676, -83.075, 50.926]
  Set speed (15.0 mm/s)
  Call Extruder(0.050)
  MoveL 9093 to (497.69, 497.21, 17.6) mm, rotated rx 0 ry 90 rz 0 deg; joints [-11.797, -28.202, 112.003, -15.809, -83.172, 50.914]
  Set speed (120.0 mm/s)
  MoveL 9094 to (497.36, 496.55, 17.6) mm, rotated rx 0 ry 90 rz 0 deg; joints [-11.743, -28.21, 112.06, -15.753, -83.216, 50.895]
  Set speed (15.0 mm/s)
  Call Extruder(0.107)
  MoveL 9095 to (499.95, 493.96, 17.6) mm, rotated rx 0 ry 90 rz 0 deg; joints [-11.455, -28.172, 111.814, -15.47, -83.008, 50.921]
  Set speed (120.0 mm/s)
  MoveL 9096 to (498.96, 493.96, 17.6) mm, rotated rx 0 ry 90 rz 0 deg; joints [-11.474, -28.191, 111.932, -15.486, -83.104, 50.896]
  Set speed (15.0 mm/s)
  Call Extruder(0.080)
  MoveL 9097 to (497.02, 495.9, 17.6) mm, rotated rx 0 ry 90 rz 0 deg; joints [-11.689, -28.219, 112.116, -15.697, -83.26, 50.877]
  Set speed (120.0 mm/s)
  MoveL 9098 to (496.69, 495.24, 17.6) mm, rotated rx 0 ry 90 rz 0 deg; joints [-11.635, -28.228, 112.172, -15.641, -83.304, 50.858]
  Set speed (15.0 mm/s)
  Call Extruder(0.053)
  MoveL 9099 to (497.97, 493.96, 17.6) mm, rotated rx 0 ry 90 rz 0 deg; joints [-11.492, -28.209, 112.05, -15.501, -83.201, 50.871]
  Set speed (120.0 mm/s)
  MoveL 9100 to (496.98, 493.96, 17.6) mm, rotated rx 0 ry 90 rz 0 deg; joints [-11.511, -28.227, 112.168, -15.517, -83.298, 50.846]
  Set speed (15.0 mm/s)
  Call Extruder(0.026)
  MoveL 9101 to (496.35, 494.59, 17.6) mm, rotated rx 0 ry 90 rz 0 deg; joints [-11.58, -28.236, 112.227, -15.585, -83.348, 50.84]
  Set speed (120.0 mm/s)
  MoveL 9102 to (499.33, 495.57, 17.6) mm, rotated rx 0 ry 90 rz 0 deg; joints [-11.614, -28.178, 111.848, -15.629, -83.04, 50.93]
  Set speed (15.0 mm/s)
  Call Extruder(0.066)
  MoveL 9103 to (500.94, 493.96, 17.6) mm, rotated rx 0 ry 90 rz 0 deg; joints [-11.437, -28.154, 111.695, -15.455, -82.911, 50.946]
  Set speed (120.0 mm/s)
  MoveL 9104 to (501.93, 493.96, 17.6) mm, rotated rx 0 ry 90 rz 0 deg; joints [-11.418, -28.135, 111.577, -15.44, -82.814, 50.971]
  Set speed (15.0 mm/s)
  MoveL 9105 to (500.32, 495.56, 17.6) mm, rotated rx 0 ry 90 rz 0 deg; joints [-11.596, -28.159, 111.73, -15.614, -82.944, 50.955]
  Set speed (120.0 mm/s)
  MoveL 9106 to (501.31, 495.57, 17.6) mm, rotated rx 0 ry 90 rz 0 deg; joints [-11.577, -28.14, 111.611, -15.599, -82.847, 50.98]
  Set speed (15.0 mm/s)
  MoveL 9107 to (502.92, 493.96, 17.6) mm, rotated rx 0 ry 90 rz 0 deg; joints [-11.4, -28.116, 111.458, -15.425, -82.718, 50.995]
  Set speed (120.0 mm/s)
  MoveL 9108 to (503.91, 493.96, 17.6) mm, rotated rx 0 ry 90 rz 0 deg; joints [-11.382, -28.097, 111.339, -15.41, -82.621, 51.02]
  Set speed (15.0 mm/s)
  MoveL 9109 to (502.3, 495.57, 17.6) mm, rotated rx 0 ry 90 rz 0 deg; joints [-11.558, -28.121, 111.493, -15.583, -82.751, 51.005]
  Set speed (120.0 mm/s)
  MoveL 9110 to (503.29, 495.57, 17.6) mm, rotated rx 0 ry 90 rz 0 deg; joints [-11.54, -28.102, 111.374, -15.568, -82.654, 51.03]
  Set speed (15.0 mm/s)
  Call Extruder(0.035)
  MoveL 9111 to (504.15, 494.7, 17.6) mm, rotated rx 0 ry 90 rz 0 deg; joints [-11.445, -28.089, 111.292, -15.475, -82.585, 51.038]
  Set speed (120.0 mm/s)
  MoveL 9112 to (502.26, 502.54, 17.6) mm, rotated rx 0 ry 90 rz 0 deg; joints [-12.196, -28.094, 111.322, -16.231, -82.634, 51.117]
  Set speed (15.0 mm/s)
  Call Extruder(0.050)
  MoveL 9113 to (501.03, 503.76, 17.6) mm, rotated rx 0 ry 90 rz 0 deg; joints [-12.332, -28.112, 111.437, -16.365, -82.73, 51.105]
  MoveL 9114 to (500.91, 503.89, 17.6) mm, rotated rx 0 ry 90 rz 0 deg; joints [-12.346, -28.114, 111.448, -16.378, -82.74, 51.104]
  Set speed (120.0 mm/s)
  MoveL 9115 to (490.68, 490.68, 17.6) mm, rotated rx 0 ry 90 rz 0 deg; joints [-11.324, -28.35, 112.995, -15.308, -83.972, 50.64]
  Set speed (1000.0 mm/s)
  MoveL 9116 to (490.68, 490.68, 17.7) mm, rotated rx 0 ry 90 rz 0 deg; joints [-11.324, -28.361, 113, -15.308, -83.966, 50.641]
  Set speed (30.0 mm/s)
  Call Extruder(0.287)
  MoveL 9117 to (497.65, 497.65, 17.7) mm, rotated rx 0 ry 90 rz 0 deg; joints [-11.838, -28.211, 112.002, -15.851, -83.162, 50.921]
  MoveL 9118 to (497.78, 497.78, 17.7) mm, rotated rx 0 ry 90 rz 0 deg; joints [-11.847, -28.209, 111.984, -15.861, -83.148, 50.926]
  Set speed (120.0 mm/s)
  MoveL 9119 to (499.24, 500.76, 17.7) mm, rotated rx 0 ry 90 rz 0 deg; joints [-12.093, -28.17, 111.734, -16.115, -82.953, 51.011]
  Set speed (30.0 mm/s)
  Call Extruder(0.352)
  MoveL 9120 to (490.68, 509.32, 17.7) mm, rotated rx 0 ry 90 rz 0 deg; joints [-13.056, -28.291, 112.524, -17.062, -83.623, 50.918]
  MoveL 9121 to (490.56, 509.44, 17.7) mm, rotated rx 0 ry 90 rz 0 deg; joints [-13.07, -28.292, 112.535, -17.076, -83.632, 50.916]
  Set speed (120.0 mm/s)
  MoveL 9122 to (496.13, 506.03, 17.7) mm, rotated rx 0 ry 90 rz 0 deg; joints [-12.639, -28.206, 111.967, -16.658, -83.159, 51.013]
  Set speed (30.0 mm/s)
  Call Extruder(0.224)
  MoveL 9123 to (490.68, 500.58, 17.7) mm, rotated rx 0 ry 90 rz 0 deg; joints [-12.247, -28.325, 112.756, -16.242, -83.789, 50.784]
  Set speed (120.0 mm/s)
  MoveL 9124 to (490.68, 499.42, 17.7) mm, rotated rx 0 ry 90 rz 0 deg; joints [-12.139, -28.329, 112.785, -16.133, -83.811, 50.766]
  Set speed (30.0 mm/s)
  Call Extruder(0.215)
  MoveL 9125 to (495.89, 494.21, 17.7) mm, rotated rx 0 ry 90 rz 0 deg; joints [-11.554, -28.257, 112.296, -15.557, -83.394, 50.824]
  Set speed (120.0 mm/s)
  MoveL 9126 to (496.37, 493.73, 17.7) mm, rotated rx 0 ry 90 rz 0 deg; joints [-11.5, -28.25, 112.251, -15.504, -83.356, 50.829]
  Set speed (30.0 mm/s)
  Call Extruder(0.125)
  MoveL 9127 to (499.42, 490.68, 17.7) mm, rotated rx 0 ry 90 rz 0 deg; joints [-11.163, -28.205, 111.96, -15.172, -83.109, 50.859]
  Set speed (120.0 mm/s)
  MoveL 9128 to (500.58, 490.68, 17.7) mm, rotated rx 0 ry 90 rz 0 deg; joints [-11.141, -28.183, 111.822, -15.155, -82.996, 50.888]
  Set speed (30.0 mm/s)
  MoveL 9129 to (503.63, 493.73, 17.7) mm, rotated rx 0 ry 90 rz 0 deg; joints [-11.366, -28.114, 111.384, -15.392, -82.647, 51.011]
  Set speed (120.0 mm/s)
  MoveL 9130 to (504.39, 494.49, 17.7) mm, rotated rx 0 ry 90 rz 0 deg; joints [-11.421, -28.096, 111.273, -15.452, -82.56, 51.042]
  Set speed (30.0 mm/s)
  Call Extruder(0.203)
  MoveL 9131 to (509.32, 499.42, 17.7) mm, rotated rx 0 ry 90 rz 0 deg; joints [-11.777, -27.977, 110.558, -15.833, -81.998, 51.247]
  Set speed (120.0 mm/s)
  MoveL 9132 to (509.32, 500.58, 17.7) mm, rotated rx 0 ry 90 rz 0 deg; joints [-11.882, -27.972, 110.529, -15.939, -81.978, 51.267]
  Set speed (30.0 mm/s)
  Call Extruder(0.212)
  MoveL 9133 to (504.16, 505.74, 17.7) mm, rotated rx 0 ry 90 rz 0 deg; joints [-12.449, -28.053, 111.016, -16.496, -82.387, 51.222]
  Set speed (120.0 mm/s)
  MoveL 9134 to (503.3, 506.6, 17.7) mm, rotated rx 0 ry 90 rz 0 deg; joints [-12.544, -28.067, 111.096, -16.589, -82.454, 51.214]
  Set speed (30.0 mm/s)
  Call Extruder(0.112)
  MoveL 9135 to (500.58, 509.32, 17.7) mm, rotated rx 0 ry 90 rz 0 deg; joints [-12.847, -28.108, 111.348, -16.887, -82.667, 51.188]
  Set speed (120.0 mm/s)
  MoveL 9136 to (499.42, 509.32, 17.7) mm, rotated rx 0 ry 90 rz 0 deg; joints [-12.872, -28.13, 111.487, -16.907, -82.779, 51.156]
  Set speed (30.0 mm/s)
  Call Extruder(0.112)
  MoveL 9137 to (496.7, 506.6, 17.7) mm, rotated rx 0 ry 90 rz 0 deg; joints [-12.679, -28.193, 111.884, -16.701, -83.093, 51.038]
  MoveL 9138 to (496.57, 506.47, 17.7) mm, rotated rx 0 ry 90 rz 0 deg; joints [-12.67, -28.196, 111.902, -16.692, -83.107, 51.033]
  Set speed (120.0 mm/s)
  MoveL 9139 to (502.51, 502.51, 17.7) mm, rotated rx 0 ry 90 rz 0 deg; joints [-12.188, -28.1, 111.299, -16.224, -82.605, 51.124]
  Set speed (30.0 mm/s)
  Call Extruder(0.280)
  MoveL 9140 to (509.32, 509.32, 17.7) mm, rotated rx 0 ry 90 rz 0 deg; joints [-12.669, -27.933, 110.3, -16.741, -81.825, 51.421]
  MoveL 9141 to (509.44, 509.44, 17.7) mm, rotated rx 0 ry 90 rz 0 deg; joints [-12.677, -27.929, 110.282, -16.75, -81.81, 51.426]
  Set speed (120.0 mm/s)
  MoveL 9142 to (500.81, 499.19, 17.7) mm, rotated rx 0 ry 90 rz 0 deg; joints [-11.919, -28.146, 111.586, -15.944, -82.828, 51.026]
  Set speed (30.0 mm/s)
  Call Extruder(0.140)
  MoveL 9143 to (504.2, 495.8, 17.7) mm, rotated rx 0 ry 90 rz 0 deg; joints [-11.544, -28.094, 111.265, -15.576, -82.557, 51.058]
  Set speed (120.0 mm/s)
  MoveL 9144 to (504.39, 495.61, 17.7) mm, rotated rx 0 ry 90 rz 0 deg; joints [-11.523, -28.091, 111.246, -15.555, -82.541, 51.06]
  Set speed (30.0 mm/s)
  Call Extruder(0.203)
  MoveL 9145 to (509.32, 490.68, 17.7) mm, rotated rx 0 ry 90 rz 0 deg; joints [-10.985, -28.013, 110.771, -15.027, -82.141, 51.101]
  MoveL 9146 to (509.44, 490.56, 17.7) mm, rotated rx 0 ry 90 rz 0 deg; joints [-10.972, -28.011, 110.759, -15.014, -82.131, 51.102]
  Set speed (120.0 mm/s)
  MoveL 9147 to (490.47, 509.53, 17.7) mm, rotated rx 0 ry 90 rz 0 deg; joints [-13.08, -28.294, 112.543, -17.085, -83.639, 50.915]
  Set speed (1000.0 mm/s)
  MoveL 9148 to (490.4, 509.6, 17.7) mm, rotated rx 0 ry 90 rz 0 deg; joints [-13.088, -28.295, 112.549, -17.093, -83.644, 50.914]
  Set speed (15.0 mm/s)
  Call Extruder(0.559)
  MoveL 9149 to (490.4, 490.4, 17.7) mm, rotated rx 0 ry 90 rz 0 deg; joints [-11.303, -28.366, 113.04, -15.286, -83.999, 50.631]
  MoveL 9150 to (509.6, 490.4, 17.7) mm, rotated rx 0 ry 90 rz 0 deg; joints [-10.955, -28.008, 110.743, -14.997, -82.118, 51.103]
  MoveL 9151 to (509.6, 509.6, 17.7) mm, rotated rx 0 ry 90 rz 0 deg; joints [-12.688, -27.925, 110.258, -16.762, -81.792, 51.433]
  MoveL 9152 to (490.4, 509.6, 17.7) mm, rotated rx 0 ry 90 rz 0 deg; joints [-13.088, -28.295, 112.549, -17.093, -83.644, 50.914]
  Set speed (120.0 mm/s)
  MoveL 9153 to (490.4, 509.2, 17.7) mm, rotated rx 0 ry 90 rz 0 deg; joints [-13.051, -28.296, 112.56, -17.056, -83.652, 50.908]
  Set speed (1000.0 mm/s)
  MoveL 9154 to (490.5, 509.2, 17.7) mm, rotated rx 0 ry 90 rz 0 deg; joints [-13.049, -28.294, 112.548, -17.054, -83.643, 50.911]
  Set speed (1000.0 mm/s)
  MoveL 9155 to (496.05, 506.68, 17.7) mm, rotated rx 0 ry 90 rz 0 deg; joints [-12.7, -28.205, 111.959, -16.72, -83.154, 51.022]
  Set speed (15.0 mm/s)
  Call Extruder(0.065)
  MoveL 9156 to (496.05, 504.44, 17.7) mm, rotated rx 0 ry 90 rz 0 deg; joints [-12.495, -28.214, 112.019, -16.512, -83.196, 50.986]
  Call Extruder(0.145)
  MoveL 9157 to (501.03, 504.44, 17.7) mm, rotated rx 0 ry 90 rz 0 deg; joints [-12.394, -28.12, 111.425, -16.428, -82.713, 51.118]
  Call Extruder(0.353)
  MoveL 9158 to (495.52, 493.65, 17.7) mm, rotated rx 0 ry 90 rz 0 deg; joints [-11.509, -28.265, 112.354, -15.51, -83.441, 50.806]
  Call Extruder(0.261)
  MoveL 9159 to (504.47, 493.65, 17.7) mm, rotated rx 0 ry 90 rz 0 deg; joints [-11.343, -28.097, 111.284, -15.372, -82.566, 51.03]
  Call Extruder(0.065)
  MoveL 9160 to (504.47, 495.88, 17.7) mm, rotated rx 0 ry 90 rz 0 deg; joints [-11.547, -28.089, 111.23, -15.579, -82.529, 51.066]
  Call Extruder(0.153)
  MoveL 9161 to (499.21, 495.88, 17.7) mm, rotated rx 0 ry 90 rz 0 deg; joints [-11.646, -28.189, 111.861, -15.661, -83.042, 50.933]
  Call Extruder(0.353)
  MoveL 9162 to (504.73, 506.68, 17.7) mm, rotated rx 0 ry 90 rz 0 deg; joints [-12.523, -28.038, 110.923, -16.573, -82.315, 51.253]
  Call Extruder(0.253)
  MoveL 9163 to (496.05, 506.68, 17.7) mm, rotated rx 0 ry 90 rz 0 deg; joints [-12.7, -28.205, 111.959, -16.72, -83.154, 51.022]
  Set speed (120.0 mm/s)
  MoveL 9164 to (496.46, 506.36, 17.7) mm, rotated rx 0 ry 90 rz 0 deg; joints [-12.662, -28.198, 111.919, -16.683, -83.12, 51.028]
  Set speed (15.0 mm/s)
  Call Extruder(0.004)
  MoveL 9165 to (496.36, 506.26, 17.7) mm, rotated rx 0 ry 90 rz 0 deg; joints [-12.655, -28.201, 111.933, -16.675, -83.132, 51.023]
  Set speed (120.0 mm/s)
  MoveL 9166 to (496.36, 505.27, 17.7) mm, rotated rx 0 ry 90 rz 0 deg; joints [-12.564, -28.205, 111.96, -16.583, -83.15, 51.007]
  Set speed (15.0 mm/s)
  Call Extruder(0.045)
  MoveL 9167 to (497.45, 506.36, 17.7) mm, rotated rx 0 ry 90 rz 0 deg; joints [-12.642, -28.18, 111.801, -16.666, -83.024, 51.054]
  Set speed (120.0 mm/s)
  MoveL 9168 to (498.44, 506.36, 17.7) mm, rotated rx 0 ry 90 rz 0 deg; joints [-12.622, -28.161, 111.683, -16.649, -82.928, 51.081]
  Set speed (15.0 mm/s)
  Call Extruder(0.066)
  MoveL 9169 to (496.84, 504.76, 17.7) mm, rotated rx 0 ry 90 rz 0 deg; joints [-12.508, -28.198, 111.916, -16.527, -83.113, 51.012]
  Set speed (120.0 mm/s)
  MoveL 9170 to (497.83, 504.76, 17.7) mm, rotated rx 0 ry 90 rz 0 deg; joints [-12.488, -28.18, 111.798, -16.511, -83.017, 51.038]
  Set speed (15.0 mm/s)
  MoveL 9171 to (499.43, 506.36, 17.7) mm, rotated rx 0 ry 90 rz 0 deg; joints [-12.602, -28.143, 111.565, -16.632, -82.833, 51.107]
  Set speed (120.0 mm/s)
  MoveL 9172 to (500.42, 506.36, 17.7) mm, rotated rx 0 ry 90 rz 0 deg; joints [-12.581, -28.124, 111.447, -16.616, -82.737, 51.134]
  Set speed (15.0 mm/s)
  MoveL 9173 to (498.82, 504.76, 17.7) mm, rotated rx 0 ry 90 rz 0 deg; joints [-12.468, -28.161, 111.68, -16.494, -82.922, 51.065]
  Set speed (120.0 mm/s)
  MoveL 9174 to (499.81, 504.76, 17.7) mm, rotated rx 0 ry 90 rz 0 deg; joints [-12.448, -28.142, 111.562, -16.477, -82.826, 51.091]
  Set speed (15.0 mm/s)
  MoveL 9175 to (501.41, 506.36, 17.7) mm, rotated rx 0 ry 90 rz 0 deg; joints [-12.561, -28.105, 111.328, -16.599, -82.641, 51.16]
  Set speed (120.0 mm/s)
  MoveL 9176 to (502.4, 506.36, 17.7) mm, rotated rx 0 ry 90 rz 0 deg; joints [-12.541, -28.085, 111.21, -16.582, -82.546, 51.186]
  Set speed (15.0 mm/s)
  MoveL 9177 to (500.8, 504.76, 17.7) mm, rotated rx 0 ry 90 rz 0 deg; joints [-12.428, -28.123, 111.444, -16.461, -82.73, 51.117]
  Set speed (120.0 mm/s)
  MoveL 9178 to (501.28, 504.25, 17.7) mm, rotated rx 0 ry 90 rz 0 deg; joints [-12.372, -28.116, 111.399, -16.406, -82.692, 51.121]
  Set speed (15.0 mm/s)
  Call Extruder(0.087)
  MoveL 9179 to (503.39, 506.36, 17.7) mm, rotated rx 0 ry 90 rz 0 deg; joints [-12.521, -28.066, 111.091, -16.566, -82.45, 51.212]
  Set speed (120.0 mm/s)
  MoveL 9180 to (504.04, 506.02, 17.7) mm, rotated rx 0 ry 90 rz 0 deg; joints [-12.477, -28.055, 111.023, -16.524, -82.393, 51.224]
  Set speed (15.0 mm/s)
  Call Extruder(0.156)
  MoveL 9181 to (500.25, 502.23, 17.7) mm, rotated rx 0 ry 90 rz 0 deg; joints [-12.208, -28.144, 111.575, -16.235, -82.828, 51.061]
  MoveL 9182 to (500.13, 502.11, 17.7) mm, rotated rx 0 ry 90 rz 0 deg; joints [-12.199, -28.147, 111.593, -16.226, -82.843, 51.056]
  Set speed (120.0 mm/s)
  MoveL 9183 to (501.96, 501.96, 17.7) mm, rotated rx 0 ry 90 rz 0 deg; joints [-12.15, -28.113, 111.378, -16.183, -82.667, 51.101]
  Set speed (15.0 mm/s)
  Call Extruder(0.155)
  MoveL 9184 to (498.19, 498.19, 17.7) mm, rotated rx 0 ry 90 rz 0 deg; joints [-11.878, -28.199, 111.924, -15.893, -83.101, 50.943]
  MoveL 9185 to (498.07, 498.07, 17.7) mm, rotated rx 0 ry 90 rz 0 deg; joints [-11.869, -28.202, 111.942, -15.883, -83.115, 50.938]
  Set speed (120.0 mm/s)
  MoveL 9186 to (499.89, 497.91, 17.7) mm, rotated rx 0 ry 90 rz 0 deg; joints [-11.819, -28.169, 111.729, -15.839, -82.94, 50.983]
  Set speed (15.0 mm/s)
  Call Extruder(0.155)
  MoveL 9187 to (496.13, 494.15, 17.7) mm, rotated rx 0 ry 90 rz 0 deg; joints [-11.544, -28.252, 112.27, -15.548, -83.372, 50.829]
  Set speed (120.0 mm/s)
  MoveL 9188 to (496.93, 493.96, 17.7) mm, rotated rx 0 ry 90 rz 0 deg; joints [-11.512, -28.239, 112.179, -15.518, -83.297, 50.847]
  Set speed (15.0 mm/s)
  Call Extruder(0.079)
  MoveL 9189 to (498.85, 495.88, 17.7) mm, rotated rx 0 ry 90 rz 0 deg; joints [-11.652, -28.196, 111.903, -15.667, -83.077, 50.924]
  Set speed (120.0 mm/s)
  MoveL 9190 to (499.52, 495.57, 17.7) mm, rotated rx 0 ry 90 rz 0 deg; joints [-11.611, -28.185, 111.83, -15.627, -83.016, 50.937]
  Set speed (15.0 mm/s)
  Call Extruder(0.066)
  MoveL 9191 to (497.92, 493.96, 17.7) mm, rotated rx 0 ry 90 rz 0 deg; joints [-11.493, -28.22, 112.061, -15.502, -83.2, 50.872]
  Set speed (120.0 mm/s)
  MoveL 9192 to (498.91, 493.96, 17.7) mm, rotated rx 0 ry 90 rz 0 deg; joints [-11.475, -28.202, 111.943, -15.487, -83.104, 50.896]
  Set speed (15.0 mm/s)
  MoveL 9193 to (500.51, 495.57, 17.7) mm, rotated rx 0 ry 90 rz 0 deg; joints [-11.592, -28.166, 111.712, -15.611, -82.92, 50.962]
  Set speed (120.0 mm/s)
  MoveL 9194 to (501.5, 495.56, 17.7) mm, rotated rx 0 ry 90 rz 0 deg; joints [-11.573, -28.147, 111.593, -15.596, -82.823, 50.987]
  Set speed (15.0 mm/s)
  MoveL 9195 to (499.9, 493.96, 17.7) mm, rotated rx 0 ry 90 rz 0 deg; joints [-11.456, -28.184, 111.824, -15.471, -83.007, 50.921]
  Set speed (120.0 mm/s)
  MoveL 9196 to (500.89, 493.96, 17.7) mm, rotated rx 0 ry 90 rz 0 deg; joints [-11.438, -28.165, 111.706, -15.456, -82.91, 50.946]
  Set speed (15.0 mm/s)
  MoveL 9197 to (502.49, 495.57, 17.7) mm, rotated rx 0 ry 90 rz 0 deg; joints [-11.555, -28.128, 111.475, -15.58, -82.727, 51.012]
  Set speed (120.0 mm/s)
  MoveL 9198 to (503.48, 495.57, 17.7) mm, rotated rx 0 ry 90 rz 0 deg; joints [-11.536, -28.109, 111.356, -15.565, -82.63, 51.036]
  Set speed (15.0 mm/s)
  MoveL 9199 to (501.88, 493.96, 17.7) mm, rotated rx 0 ry 90 rz 0 deg; joints [-11.419, -28.146, 111.587, -15.441, -82.814, 50.971]
  Set speed (120.0 mm/s)
  MoveL 9200 to (502.87, 493.96, 17.7) mm, rotated rx 0 ry 90 rz 0 deg; joints [-11.401, -28.127, 111.469, -15.426, -82.717, 50.996]
  Set speed (15.0 mm/s)
  Call Extruder(0.053)
  MoveL 9201 to (504.16, 495.25, 17.7) mm, rotated rx 0 ry 90 rz 0 deg; joints [-11.495, -28.097, 111.283, -15.525, -82.57, 51.048]
  Set speed (120.0 mm/s)
  MoveL 9202 to (504.16, 494.26, 17.7) mm, rotated rx 0 ry 90 rz 0 deg; joints [-11.404, -28.101, 111.307, -15.434, -82.587, 51.032]
  Set speed (15.0 mm/s)
  Call Extruder(0.012)
  MoveL 9203 to (503.86, 493.96, 17.7) mm, rotated rx 0 ry 90 rz 0 deg; joints [-11.383, -28.108, 111.35, -15.411, -82.62, 51.02]
  Set speed (120.0 mm/s)
  MoveL 9204 to (500.93, 499.94, 17.7) mm, rotated rx 0 ry 90 rz 0 deg; joints [-11.985, -28.141, 111.553, -16.011, -82.804, 51.041]
  Set speed (15.0 mm/s)
  Call Extruder(0.155)
  MoveL 9205 to (497.16, 496.17, 17.7) mm, rotated rx 0 ry 90 rz 0 deg; joints [-11.711, -28.226, 112.097, -15.721, -83.237, 50.886]
  MoveL 9206 to (497.04, 496.05, 17.7) mm, rotated rx 0 ry 90 rz 0 deg; joints [-11.702, -28.229, 112.115, -15.711, -83.251, 50.881]
  Set speed (120.0 mm/s)
  MoveL 9207 to (499.22, 500.21, 17.7) mm, rotated rx 0 ry 90 rz 0 deg; joints [-12.043, -28.172, 111.75, -16.064, -82.965, 51.002]
  Set speed (15.0 mm/s)
  Call Extruder(0.156)
  MoveL 9208 to (503, 503.99, 17.7) mm, rotated rx 0 ry 90 rz 0 deg; joints [-12.314, -28.084, 111.201, -16.354, -82.53, 51.162]
  MoveL 9209 to (503.12, 504.12, 17.7) mm, rotated rx 0 ry 90 rz 0 deg; joints [-12.323, -28.081, 111.183, -16.363, -82.516, 51.167]
  Set speed (120.0 mm/s)
  MoveL 9210 to (490.68, 490.68, 17.7) mm, rotated rx 0 ry 90 rz 0 deg; joints [-11.324, -28.361, 113, -15.308, -83.966, 50.641]
  Set speed (1000.0 mm/s)
  MoveL 9211 to (490.68, 490.68, 17.8) mm, rotated rx 0 ry 90 rz 0 deg; joints [-11.324, -28.371, 113.005, -15.308, -83.961, 50.643]
  Set speed (30.0 mm/s)
  Call Extruder(0.287)
  MoveL 9212 to (497.65, 497.65, 17.8) mm, rotated rx 0 ry 90 rz 0 deg; joints [-11.838, -28.222, 112.007, -15.851, -83.157, 50.923]
  MoveL 9213 to (497.78, 497.78, 17.8) mm, rotated rx 0 ry 90 rz 0 deg; joints [-11.847, -28.219, 111.989, -15.861, -83.143, 50.928]
  Set speed (120.0 mm/s)
  MoveL 9214 to (499.24, 500.76, 17.8) mm, rotated rx 0 ry 90 rz 0 deg; joints [-12.093, -28.18, 111.739, -16.116, -82.948, 51.013]
  Set speed (30.0 mm/s)
  Call Extruder(0.352)
  MoveL 9215 to (490.68, 509.32, 17.8) mm, rotated rx 0 ry 90 rz 0 deg; joints [-13.056, -28.301, 112.529, -17.062, -83.618, 50.919]
  MoveL 9216 to (490.56, 509.44, 17.8) mm, rotated rx 0 ry 90 rz 0 deg; joints [-13.07, -28.303, 112.54, -17.076, -83.627, 50.918]
  Set speed (120.0 mm/s)
  MoveL 9217 to (496.13, 506.03, 17.8) mm, rotated rx 0 ry 90 rz 0 deg; joints [-12.639, -28.217, 111.972, -16.658, -83.154, 51.015]
  Set speed (30.0 mm/s)
  Call Extruder(0.224)
  MoveL 9218 to (490.68, 500.58, 17.8) mm, rotated rx 0 ry 90 rz 0 deg; joints [-12.247, -28.336, 112.761, -16.242, -83.784, 50.785]
  Set speed (120.0 mm/s)
  MoveL 9219 to (490.68, 499.42, 17.8) mm, rotated rx 0 ry 90 rz 0 deg; joints [-12.139, -28.34, 112.79, -16.133, -83.805, 50.768]
  Set speed (30.0 mm/s)
  Call Extruder(0.215)
  MoveL 9220 to (495.89, 494.21, 17.8) mm, rotated rx 0 ry 90 rz 0 deg; joints [-11.554, -28.267, 112.302, -15.557, -83.389, 50.825]
  Set speed (120.0 mm/s)
  MoveL 9221 to (496.37, 493.73, 17.8) mm, rotated rx 0 ry 90 rz 0 deg; joints [-11.5, -28.26, 112.256, -15.505, -83.351, 50.83]
  Set speed (30.0 mm/s)
  Call Extruder(0.125)
  MoveL 9222 to (499.42, 490.68, 17.8) mm, rotated rx 0 ry 90 rz 0 deg; joints [-11.163, -28.216, 111.965, -15.172, -83.104, 50.861]
  Set speed (120.0 mm/s)
  MoveL 9223 to (500.58, 490.68, 17.8) mm, rotated rx 0 ry 90 rz 0 deg; joints [-11.141, -28.194, 111.827, -15.155, -82.99, 50.89]
  Set speed (30.0 mm/s)
  MoveL 9224 to (503.63, 493.73, 17.8) mm, rotated rx 0 ry 90 rz 0 deg; joints [-11.366, -28.124, 111.389, -15.393, -82.642, 51.012]
  Set speed (120.0 mm/s)
  MoveL 9225 to (504.39, 494.49, 17.8) mm, rotated rx 0 ry 90 rz 0 deg; joints [-11.421, -28.106, 111.279, -15.452, -82.554, 51.043]
  Set speed (30.0 mm/s)
  Call Extruder(0.203)
  MoveL 9226 to (509.32, 499.42, 17.8) mm, rotated rx 0 ry 90 rz 0 deg; joints [-11.777, -27.987, 110.563, -15.833, -81.992, 51.248]
  Set speed (120.0 mm/s)
  MoveL 9227 to (509.32, 500.58, 17.8) mm, rotated rx 0 ry 90 rz 0 deg; joints [-11.882, -27.982, 110.534, -15.939, -81.973, 51.268]
  Set speed (30.0 mm/s)
  Call Extruder(0.212)
  MoveL 9228 to (504.16, 505.74, 17.8) mm, rotated rx 0 ry 90 rz 0 deg; joints [-12.449, -28.064, 111.021, -16.496, -82.382, 51.223]
  Set speed (120.0 mm/s)
  MoveL 9229 to (503.3, 506.6, 17.8) mm, rotated rx 0 ry 90 rz 0 deg; joints [-12.544, -28.077, 111.101, -16.589, -82.449, 51.215]
  Set speed (30.0 mm/s)
  Call Extruder(0.112)
  MoveL 9230 to (500.58, 509.32, 17.8) mm, rotated rx 0 ry 90 rz 0 deg; joints [-12.847, -28.118, 111.353, -16.887, -82.662, 51.189]
  Set speed (120.0 mm/s)
  MoveL 9231 to (499.42, 509.32, 17.8) mm, rotated rx 0 ry 90 rz 0 deg; joints [-12.872, -28.141, 111.492, -16.907, -82.774, 51.158]
  Set speed (30.0 mm/s)
  Call Extruder(0.112)
  MoveL 9232 to (496.7, 506.6, 17.8) mm, rotated rx 0 ry 90 rz 0 deg; joints [-12.679, -28.204, 111.889, -16.701, -83.088, 51.039]
  MoveL 9233 to (496.57, 506.47, 17.8) mm, rotated rx 0 ry 90 rz 0 deg; joints [-12.67, -28.206, 111.907, -16.692, -83.102, 51.034]
  Set speed (120.0 mm/s)
  MoveL 9234 to (502.51, 502.51, 17.8) mm, rotated rx 0 ry 90 rz 0 deg; joints [-12.188, -28.11, 111.304, -16.224, -82.6, 51.126]
  Set speed (30.0 mm/s)
  Call Extruder(0.280)
  MoveL 9235 to (509.32, 509.32, 17.8) mm, rotated rx 0 ry 90 rz 0 deg; joints [-12.669, -27.943, 110.305, -16.741, -81.819, 51.422]
  MoveL 9236 to (509.44, 509.44, 17.8) mm, rotated rx 0 ry 90 rz 0 deg; joints [-12.677, -27.94, 110.287, -16.75, -81.805, 51.428]
  Set speed (120.0 mm/s)
  MoveL 9237 to (500.81, 499.19, 17.8) mm, rotated rx 0 ry 90 rz 0 deg; joints [-11.919, -28.157, 111.592, -15.944, -82.823, 51.028]
  Set speed (30.0 mm/s)
  Call Extruder(0.140)
  MoveL 9238 to (504.2, 495.8, 17.8) mm, rotated rx 0 ry 90 rz 0 deg; joints [-11.544, -28.105, 111.27, -15.576, -82.551, 51.06]
  Set speed (120.0 mm/s)
  MoveL 9239 to (504.39, 495.61, 17.8) mm, rotated rx 0 ry 90 rz 0 deg; joints [-11.523, -28.102, 111.251, -15.556, -82.536, 51.061]
  Set speed (30.0 mm/s)
  Call Extruder(0.203)
  MoveL 9240 to (509.32, 490.68, 17.8) mm, rotated rx 0 ry 90 rz 0 deg; joints [-10.985, -28.023, 110.776, -15.027, -82.136, 51.103]
  MoveL 9241 to (509.44, 490.56, 17.8) mm, rotated rx 0 ry 90 rz 0 deg; joints [-10.972, -28.021, 110.764, -15.014, -82.126, 51.104]
  Set speed (120.0 mm/s)
  MoveL 9242 to (490.47, 509.53, 17.8) mm, rotated rx 0 ry 90 rz 0 deg; joints [-13.08, -28.304, 112.548, -17.086, -83.634, 50.917]
  Set speed (1000.0 mm/s)
  MoveL 9243 to (490.4, 509.6, 17.8) mm, rotated rx 0 ry 90 rz 0 deg; joints [-13.088, -28.305, 112.554, -17.093, -83.639, 50.916]
  Set speed (15.0 mm/s)
  Call Extruder(0.559)
  MoveL 9244 to (490.4, 490.4, 17.8) mm, rotated rx 0 ry 90 rz 0 deg; joints [-11.303, -28.377, 113.045, -15.286, -83.993, 50.632]
  MoveL 9245 to (509.6, 490.4, 17.8) mm, rotated rx 0 ry 90 rz 0 deg; joints [-10.955, -28.019, 110.748, -14.997, -82.113, 51.105]
  MoveL 9246 to (509.6, 509.6, 17.8) mm, rotated rx 0 ry 90 rz 0 deg; joints [-12.688, -27.936, 110.263, -16.762, -81.787, 51.435]
  MoveL 9247 to (490.4, 509.6, 17.8) mm, rotated rx 0 ry 90 rz 0 deg; joints [-13.088, -28.305, 112.554, -17.093, -83.639, 50.916]
  Set speed (120.0 mm/s)
  MoveL 9248 to (490.4, 509.2, 17.8) mm, rotated rx 0 ry 90 rz 0 deg; joints [-13.051, -28.307, 112.565, -17.056, -83.647, 50.91]
  Set speed (1000.0 mm/s)
  MoveL 9249 to (490.5, 509.2, 17.8) mm, rotated rx 0 ry 90 rz 0 deg; joints [-13.049, -28.305, 112.553, -17.054, -83.637, 50.912]
  Set speed (1000.0 mm/s)
  MoveL 9250 to (496.05, 506.68, 17.8) mm, rotated rx 0 ry 90 rz 0 deg; joints [-12.7, -28.215, 111.965, -16.72, -83.149, 51.023]
  Set speed (15.0 mm/s)
  Call Extruder(0.065)
  MoveL 9251 to (496.05, 504.45, 17.8) mm, rotated rx 0 ry 90 rz 0 deg; joints [-12.495, -28.225, 112.024, -16.512, -83.191, 50.987]
  Call Extruder(0.145)
  MoveL 9252 to (501.03, 504.45, 17.8) mm, rotated rx 0 ry 90 rz 0 deg; joints [-12.394, -28.131, 111.43, -16.428, -82.708, 51.119]
  Call Extruder(0.353)
  MoveL 9253 to (495.52, 493.65, 17.8) mm, rotated rx 0 ry 90 rz 0 deg; joints [-11.509, -28.276, 112.359, -15.511, -83.435, 50.808]
  Call Extruder(0.261)
  MoveL 9254 to (504.47, 493.65, 17.8) mm, rotated rx 0 ry 90 rz 0 deg; joints [-11.343, -28.108, 111.289, -15.373, -82.561, 51.032]
  Call Extruder(0.065)
  MoveL 9255 to (504.47, 495.88, 17.8) mm, rotated rx 0 ry 90 rz 0 deg; joints [-11.547, -28.099, 111.235, -15.58, -82.523, 51.068]
  Call Extruder(0.153)
  MoveL 9256 to (499.21, 495.88, 17.8) mm, rotated rx 0 ry 90 rz 0 deg; joints [-11.646, -28.2, 111.866, -15.661, -83.037, 50.935]
  Call Extruder(0.353)
  MoveL 9257 to (504.73, 506.68, 17.8) mm, rotated rx 0 ry 90 rz 0 deg; joints [-12.523, -28.048, 110.928, -16.573, -82.31, 51.255]
  Call Extruder(0.253)
  MoveL 9258 to (496.05, 506.68, 17.8) mm, rotated rx 0 ry 90 rz 0 deg; joints [-12.7, -28.215, 111.965, -16.72, -83.149, 51.023]
  Set speed (120.0 mm/s)
  MoveL 9259 to (503.93, 505.81, 17.8) mm, rotated rx 0 ry 90 rz 0 deg; joints [-12.461, -28.068, 111.046, -16.507, -82.402, 51.219]
  Set speed (15.0 mm/s)
  Call Extruder(0.023)
  MoveL 9260 to (503.39, 506.36, 17.8) mm, rotated rx 0 ry 90 rz 0 deg; joints [-12.521, -28.077, 111.097, -16.566, -82.445, 51.214]
  Set speed (120.0 mm/s)
  MoveL 9261 to (502.4, 506.36, 17.8) mm, rotated rx 0 ry 90 rz 0 deg; joints [-12.541, -28.096, 111.216, -16.583, -82.541, 51.188]
  Set speed (15.0 mm/s)
  Call Extruder(0.049)
  MoveL 9262 to (503.6, 505.16, 17.8) mm, rotated rx 0 ry 90 rz 0 deg; joints [-12.408, -28.078, 111.103, -16.452, -82.446, 51.199]
  Set speed (120.0 mm/s)
  MoveL 9263 to (503.26, 504.5, 17.8) mm, rotated rx 0 ry 90 rz 0 deg; joints [-12.355, -28.087, 111.161, -16.397, -82.49, 51.179]
  Set speed (15.0 mm/s)
  Call Extruder(0.076)
  MoveL 9264 to (501.41, 506.36, 17.8) mm, rotated rx 0 ry 90 rz 0 deg; joints [-12.561, -28.115, 111.334, -16.599, -82.637, 51.161]
  Set speed (120.0 mm/s)
  MoveL 9265 to (500.42, 506.36, 17.8) mm, rotated rx 0 ry 90 rz 0 deg; joints [-12.581, -28.134, 111.452, -16.616, -82.732, 51.135]
  Set speed (15.0 mm/s)
  Call Extruder(0.103)
  MoveL 9266 to (502.93, 503.85, 17.8) mm, rotated rx 0 ry 90 rz 0 deg; joints [-12.302, -28.096, 111.218, -16.342, -82.535, 51.159]
  Set speed (120.0 mm/s)
  MoveL 9267 to (502.59, 503.19, 17.8) mm, rotated rx 0 ry 90 rz 0 deg; joints [-12.249, -28.106, 111.275, -16.287, -82.579, 51.14]
  Set speed (15.0 mm/s)
  Call Extruder(0.050)
  MoveL 9268 to (501.37, 504.42, 17.8) mm, rotated rx 0 ry 90 rz 0 deg; joints [-12.385, -28.124, 111.39, -16.42, -82.675, 51.128]
  Set speed (120.0 mm/s)
  MoveL 9269 to (501.03, 504.76, 17.8) mm, rotated rx 0 ry 90 rz 0 deg; joints [-12.423, -28.129, 111.422, -16.457, -82.702, 51.125]
  Set speed (15.0 mm/s)
  Call Extruder(0.066)
  MoveL 9270 to (499.43, 506.36, 17.8) mm, rotated rx 0 ry 90 rz 0 deg; joints [-12.602, -28.153, 111.571, -16.633, -82.828, 51.109]
  Set speed (120.0 mm/s)
  MoveL 9271 to (498.44, 506.36, 17.8) mm, rotated rx 0 ry 90 rz 0 deg; joints [-12.622, -28.172, 111.689, -16.649, -82.924, 51.082]
  Set speed (15.0 mm/s)
  MoveL 9272 to (500.04, 504.76, 17.8) mm, rotated rx 0 ry 90 rz 0 deg; joints [-12.443, -28.148, 111.54, -16.474, -82.798, 51.098]
  Set speed (120.0 mm/s)
  MoveL 9273 to (499.05, 504.76, 17.8) mm, rotated rx 0 ry 90 rz 0 deg; joints [-12.463, -28.167, 111.658, -16.49, -82.894, 51.072]
  Set speed (15.0 mm/s)
  MoveL 9274 to (497.45, 506.36, 17.8) mm, rotated rx 0 ry 90 rz 0 deg; joints [-12.642, -28.191, 111.807, -16.666, -83.02, 51.056]
  Set speed (120.0 mm/s)
  MoveL 9275 to (496.46, 506.36, 17.8) mm, rotated rx 0 ry 90 rz 0 deg; joints [-12.663, -28.209, 111.924, -16.683, -83.115, 51.029]
  Set speed (15.0 mm/s)
  MoveL 9276 to (498.06, 504.76, 17.8) mm, rotated rx 0 ry 90 rz 0 deg; joints [-12.483, -28.186, 111.776, -16.507, -82.99, 51.046]
  Set speed (120.0 mm/s)
  MoveL 9277 to (497.07, 504.76, 17.8) mm, rotated rx 0 ry 90 rz 0 deg; joints [-12.503, -28.204, 111.894, -16.524, -83.086, 51.02]
  Set speed (15.0 mm/s)
  Call Extruder(0.029)
  MoveL 9278 to (496.36, 505.47, 17.8) mm, rotated rx 0 ry 90 rz 0 deg; joints [-12.583, -28.215, 111.959, -16.602, -83.141, 51.012]
  Set speed (120.0 mm/s)
  MoveL 9279 to (500.7, 503.11, 17.8) mm, rotated rx 0 ry 90 rz 0 deg; joints [-12.279, -28.143, 111.504, -16.31, -82.764, 51.089]
  Set speed (15.0 mm/s)
  Call Extruder(0.050)
  MoveL 9280 to (501.92, 501.89, 17.8) mm, rotated rx 0 ry 90 rz 0 deg; joints [-12.143, -28.124, 111.39, -16.176, -82.667, 51.1]
  Set speed (120.0 mm/s)
  MoveL 9281 to (501.59, 501.23, 17.8) mm, rotated rx 0 ry 90 rz 0 deg; joints [-12.09, -28.133, 111.446, -16.121, -82.711, 51.081]
  Set speed (15.0 mm/s)
  MoveL 9282 to (500.37, 502.45, 17.8) mm, rotated rx 0 ry 90 rz 0 deg; joints [-12.226, -28.152, 111.561, -16.254, -82.808, 51.069]
  Set speed (120.0 mm/s)
  MoveL 9283 to (500.03, 501.8, 17.8) mm, rotated rx 0 ry 90 rz 0 deg; joints [-12.172, -28.161, 111.618, -16.199, -82.852, 51.05]
  Set speed (15.0 mm/s)
  Call Extruder(0.050)
  MoveL 9284 to (501.25, 500.58, 17.8) mm, rotated rx 0 ry 90 rz 0 deg; joints [-12.037, -28.143, 111.503, -16.066, -82.755, 51.062]
  Set speed (120.0 mm/s)
  MoveL 9285 to (500.92, 499.92, 17.8) mm, rotated rx 0 ry 90 rz 0 deg; joints [-11.983, -28.152, 111.56, -16.01, -82.8, 51.042]
  Set speed (15.0 mm/s)
  Call Extruder(0.050)
  MoveL 9286 to (499.7, 501.14, 17.8) mm, rotated rx 0 ry 90 rz 0 deg; joints [-12.119, -28.17, 111.675, -16.143, -82.897, 51.031]
  Set speed (120.0 mm/s)
  MoveL 9287 to (499.36, 500.49, 17.8) mm, rotated rx 0 ry 90 rz 0 deg; joints [-12.066, -28.179, 111.731, -16.088, -82.941, 51.011]
  Set speed (15.0 mm/s)
  Call Extruder(0.050)
  MoveL 9288 to (500.58, 499.27, 17.8) mm, rotated rx 0 ry 90 rz 0 deg; joints [-11.93, -28.161, 111.617, -15.955, -82.844, 51.023]
  Set speed (120.0 mm/s)
  MoveL 9289 to (500.25, 498.61, 17.8) mm, rotated rx 0 ry 90 rz 0 deg; joints [-11.876, -28.17, 111.673, -15.899, -82.888, 51.004]
  Set speed (15.0 mm/s)
  MoveL 9290 to (499.03, 499.83, 17.8) mm, rotated rx 0 ry 90 rz 0 deg; joints [-12.012, -28.188, 111.788, -16.032, -82.985, 50.992]
  Set speed (120.0 mm/s)
  MoveL 9291 to (498.69, 499.17, 17.8) mm, rotated rx 0 ry 90 rz 0 deg; joints [-11.958, -28.197, 111.845, -15.977, -83.029, 50.973]
  Set speed (15.0 mm/s)
  Call Extruder(0.050)
  MoveL 9292 to (499.91, 497.96, 17.8) mm, rotated rx 0 ry 90 rz 0 deg; joints [-11.823, -28.179, 111.73, -15.844, -82.932, 50.985]
  Set speed (120.0 mm/s)
  MoveL 9293 to (499.58, 497.3, 17.8) mm, rotated rx 0 ry 90 rz 0 deg; joints [-11.769, -28.187, 111.786, -15.788, -82.976, 50.966]
  Set speed (15.0 mm/s)
  MoveL 9294 to (498.36, 498.52, 17.8) mm, rotated rx 0 ry 90 rz 0 deg; joints [-11.905, -28.205, 111.901, -15.921, -83.073, 50.954]
  Set speed (120.0 mm/s)
  MoveL 9295 to (498.03, 497.86, 17.8) mm, rotated rx 0 ry 90 rz 0 deg; joints [-11.851, -28.214, 111.957, -15.865, -83.117, 50.936]
  Set speed (15.0 mm/s)
  Call Extruder(0.050)
  MoveL 9296 to (499.24, 496.65, 17.8) mm, rotated rx 0 ry 90 rz 0 deg; joints [-11.715, -28.196, 111.842, -15.732, -83.02, 50.948]
  Set speed (120.0 mm/s)
  MoveL 9297 to (498.91, 495.99, 17.8) mm, rotated rx 0 ry 90 rz 0 deg; joints [-11.662, -28.205, 111.899, -15.676, -83.064, 50.929]
  Set speed (15.0 mm/s)
  Call Extruder(0.050)
  MoveL 9298 to (497.69, 497.21, 17.8) mm, rotated rx 0 ry 90 rz 0 deg; joints [-11.797, -28.223, 112.014, -15.809, -83.161, 50.917]
  Set speed (120.0 mm/s)
  MoveL 9299 to (497.36, 496.55, 17.8) mm, rotated rx 0 ry 90 rz 0 deg; joints [-11.743, -28.232, 112.07, -15.754, -83.205, 50.898]
  Set speed (15.0 mm/s)
  Call Extruder(0.107)
  MoveL 9300 to (499.95, 493.96, 17.8) mm, rotated rx 0 ry 90 rz 0 deg; joints [-11.455, -28.193, 111.824, -15.471, -82.997, 50.924]
  Set speed (120.0 mm/s)
  MoveL 9301 to (498.96, 493.96, 17.8) mm, rotated rx 0 ry 90 rz 0 deg; joints [-11.474, -28.212, 111.942, -15.486, -83.094, 50.899]
  Set speed (15.0 mm/s)
  Call Extruder(0.080)
  MoveL 9302 to (497.02, 495.9, 17.8) mm, rotated rx 0 ry 90 rz 0 deg; joints [-11.689, -28.24, 112.126, -15.698, -83.25, 50.88]
  Set speed (120.0 mm/s)
  MoveL 9303 to (496.69, 495.24, 17.8) mm, rotated rx 0 ry 90 rz 0 deg; joints [-11.635, -28.249, 112.182, -15.642, -83.294, 50.861]
  Set speed (15.0 mm/s)
  Call Extruder(0.053)
  MoveL 9304 to (497.97, 493.96, 17.8) mm, rotated rx 0 ry 90 rz 0 deg; joints [-11.492, -28.23, 112.06, -15.502, -83.191, 50.874]
  Set speed (120.0 mm/s)
  MoveL 9305 to (496.98, 493.96, 17.8) mm, rotated rx 0 ry 90 rz 0 deg; joints [-11.511, -28.248, 112.178, -15.517, -83.287, 50.849]
  Set speed (15.0 mm/s)
  Call Extruder(0.026)
  MoveL 9306 to (496.35, 494.59, 17.8) mm, rotated rx 0 ry 90 rz 0 deg; joints [-11.58, -28.257, 112.238, -15.585, -83.338, 50.843]
  Set speed (120.0 mm/s)
  MoveL 9307 to (499.33, 495.57, 17.8) mm, rotated rx 0 ry 90 rz 0 deg; joints [-11.614, -28.199, 111.858, -15.63, -83.03, 50.933]
  Set speed (15.0 mm/s)
  Call Extruder(0.066)
  MoveL 9308 to (500.94, 493.96, 17.8) mm, rotated rx 0 ry 90 rz 0 deg; joints [-11.437, -28.175, 111.705, -15.455, -82.9, 50.949]
  Set speed (120.0 mm/s)
  MoveL 9309 to (501.93, 493.96, 17.8) mm, rotated rx 0 ry 90 rz 0 deg; joints [-11.418, -28.156, 111.587, -15.44, -82.804, 50.974]
  Set speed (15.0 mm/s)
  MoveL 9310 to (500.32, 495.57, 17.8) mm, rotated rx 0 ry 90 rz 0 deg; joints [-11.596, -28.18, 111.74, -15.614, -82.933, 50.958]
  Set speed (120.0 mm/s)
  MoveL 9311 to (501.31, 495.57, 17.8) mm, rotated rx 0 ry 90 rz 0 deg; joints [-11.577, -28.161, 111.621, -15.599, -82.837, 50.983]
  Set speed (15.0 mm/s)
  MoveL 9312 to (502.92, 493.96, 17.8) mm, rotated rx 0 ry 90 rz 0 deg; joints [-11.4, -28.137, 111.468, -15.425, -82.707, 50.998]
  Set speed (120.0 mm/s)
  MoveL 9313 to (503.91, 493.96, 17.8) mm, rotated rx 0 ry 90 rz 0 deg; joints [-11.382, -28.118, 111.35, -15.41, -82.611, 51.023]
  Set speed (15.0 mm/s)
  MoveL 9314 to (502.3, 495.56, 17.8) mm, rotated rx 0 ry 90 rz 0 deg; joints [-11.558, -28.142, 111.503, -15.584, -82.74, 51.008]
  Set speed (120.0 mm/s)
  MoveL 9315 to (503.29, 495.56, 17.8) mm, rotated rx 0 ry 90 rz 0 deg; joints [-11.54, -28.123, 111.384, -15.568, -82.644, 51.033]
  Set speed (15.0 mm/s)
  Call Extruder(0.035)
  MoveL 9316 to (504.15, 494.7, 17.8) mm, rotated rx 0 ry 90 rz 0 deg; joints [-11.445, -28.11, 111.302, -15.475, -82.574, 51.041]
  Set speed (120.0 mm/s)
  MoveL 9317 to (502.26, 502.54, 17.8) mm, rotated rx 0 ry 90 rz 0 deg; joints [-12.196, -28.115, 111.333, -16.232, -82.623, 51.12]
  Set speed (15.0 mm/s)
  Call Extruder(0.050)
  MoveL 9318 to (501.03, 503.76, 17.8) mm, rotated rx 0 ry 90 rz 0 deg; joints [-12.332, -28.133, 111.447, -16.365, -82.72, 51.108]
  MoveL 9319 to (500.91, 503.89, 17.8) mm, rotated rx 0 ry 90 rz 0 deg; joints [-12.346, -28.135, 111.459, -16.378, -82.729, 51.107]
  Set speed (120.0 mm/s)
  MoveL 9320 to (490.68, 490.68, 17.8) mm, rotated rx 0 ry 90 rz 0 deg; joints [-11.324, -28.371, 113.005, -15.308, -83.961, 50.643]
  Set speed (1000.0 mm/s)
  MoveL 9321 to (490.68, 490.68, 17.9) mm, rotated rx 0 ry 90 rz 0 deg; joints [-11.324, -28.382, 113.01, -15.308, -83.956, 50.644]
  Set speed (30.0 mm/s)
  Call Extruder(0.287)
  MoveL 9322 to (497.65, 497.65, 17.9) mm, rotated rx 0 ry 90 rz 0 deg; joints [-11.838, -28.233, 112.012, -15.852, -83.152, 50.924]
  MoveL 9323 to (497.78, 497.78, 17.9) mm, rotated rx 0 ry 90 rz 0 deg; joints [-11.847, -28.23, 111.994, -15.861, -83.138, 50.929]
  Set speed (120.0 mm/s)
  MoveL 9324 to (499.24, 500.76, 17.9) mm, rotated rx 0 ry 90 rz 0 deg; joints [-12.093, -28.191, 111.744, -16.116, -82.943, 51.014]
  Set speed (30.0 mm/s)
  Call Extruder(0.352)
  MoveL 9325 to (490.68, 509.32, 17.9) mm, rotated rx 0 ry 90 rz 0 deg; joints [-13.056, -28.312, 112.534, -17.062, -83.612, 50.921]
  MoveL 9326 to (490.56, 509.44, 17.9) mm, rotated rx 0 ry 90 rz 0 deg; joints [-13.07, -28.314, 112.545, -17.076, -83.622, 50.919]
  Set speed (120.0 mm/s)
  MoveL 9327 to (496.13, 506.03, 17.9) mm, rotated rx 0 ry 90 rz 0 deg; joints [-12.639, -28.227, 111.978, -16.658, -83.148, 51.016]
  Set speed (30.0 mm/s)
  Call Extruder(0.224)
  MoveL 9328 to (490.68, 500.58, 17.9) mm, rotated rx 0 ry 90 rz 0 deg; joints [-12.247, -28.346, 112.766, -16.242, -83.779, 50.787]
  Set speed (120.0 mm/s)
  MoveL 9329 to (490.68, 499.42, 17.9) mm, rotated rx 0 ry 90 rz 0 deg; joints [-12.139, -28.351, 112.796, -16.133, -83.8, 50.77]
  Set speed (30.0 mm/s)
  Call Extruder(0.215)
  MoveL 9330 to (495.89, 494.21, 17.9) mm, rotated rx 0 ry 90 rz 0 deg; joints [-11.554, -28.278, 112.307, -15.557, -83.384, 50.827]
  Set speed (120.0 mm/s)
  MoveL 9331 to (496.37, 493.73, 17.9) mm, rotated rx 0 ry 90 rz 0 deg; joints [-11.5, -28.271, 112.261, -15.505, -83.345, 50.832]
  Set speed (30.0 mm/s)
  Call Extruder(0.125)
  MoveL 9332 to (499.42, 490.68, 17.9) mm, rotated rx 0 ry 90 rz 0 deg; joints [-11.163, -28.226, 111.971, -15.172, -83.099, 50.862]
  Set speed (120.0 mm/s)
  MoveL 9333 to (500.58, 490.68, 17.9) mm, rotated rx 0 ry 90 rz 0 deg; joints [-11.141, -28.204, 111.832, -15.155, -82.985, 50.891]
  Set speed (30.0 mm/s)
  MoveL 9334 to (503.63, 493.73, 17.9) mm, rotated rx 0 ry 90 rz 0 deg; joints [-11.366, -28.135, 111.394, -15.393, -82.637, 51.014]
  Set speed (120.0 mm/s)
  MoveL 9335 to (504.39, 494.49, 17.9) mm, rotated rx 0 ry 90 rz 0 deg; joints [-11.421, -28.117, 111.284, -15.452, -82.549, 51.045]
  Set speed (30.0 mm/s)
  Call Extruder(0.203)
  MoveL 9336 to (509.32, 499.42, 17.9) mm, rotated rx 0 ry 90 rz 0 deg; joints [-11.777, -27.998, 110.568, -15.833, -81.987, 51.25]
  Set speed (120.0 mm/s)
  MoveL 9337 to (509.32, 500.58, 17.9) mm, rotated rx 0 ry 90 rz 0 deg; joints [-11.882, -27.993, 110.539, -15.94, -81.967, 51.27]
  Set speed (30.0 mm/s)
  Call Extruder(0.212)
  MoveL 9338 to (504.16, 505.74, 17.9) mm, rotated rx 0 ry 90 rz 0 deg; joints [-12.449, -28.074, 111.026, -16.496, -82.376, 51.225]
  Set speed (120.0 mm/s)
  MoveL 9339 to (503.3, 506.6, 17.9) mm, rotated rx 0 ry 90 rz 0 deg; joints [-12.544, -28.088, 111.106, -16.59, -82.444, 51.217]
  Set speed (30.0 mm/s)
  Call Extruder(0.112)
  MoveL 9340 to (500.58, 509.32, 17.9) mm, rotated rx 0 ry 90 rz 0 deg; joints [-12.847, -28.129, 111.358, -16.887, -82.656, 51.191]
  Set speed (120.0 mm/s)
  MoveL 9341 to (499.42, 509.32, 17.9) mm, rotated rx 0 ry 90 rz 0 deg; joints [-12.872, -28.151, 111.497, -16.907, -82.768, 51.159]
  Set speed (30.0 mm/s)
  Call Extruder(0.112)
  MoveL 9342 to (496.7, 506.6, 17.9) mm, rotated rx 0 ry 90 rz 0 deg; joints [-12.679, -28.214, 111.894, -16.701, -83.082, 51.041]
  MoveL 9343 to (496.57, 506.47, 17.9) mm, rotated rx 0 ry 90 rz 0 deg; joints [-12.67, -28.217, 111.912, -16.692, -83.097, 51.036]
  Set speed (120.0 mm/s)
  MoveL 9344 to (502.51, 502.51, 17.9) mm, rotated rx 0 ry 90 rz 0 deg; joints [-12.188, -28.121, 111.309, -16.225, -82.594, 51.127]
  Set speed (30.0 mm/s)
  Call Extruder(0.280)
  MoveL 9345 to (509.32, 509.32, 17.9) mm, rotated rx 0 ry 90 rz 0 deg; joints [-12.669, -27.953, 110.31, -16.741, -81.814, 51.424]
  MoveL 9346 to (509.44, 509.44, 17.9) mm, rotated rx 0 ry 90 rz 0 deg; joints [-12.677, -27.95, 110.292, -16.751, -81.8, 51.429]
  Set speed (120.0 mm/s)
  MoveL 9347 to (500.81, 499.19, 17.9) mm, rotated rx 0 ry 90 rz 0 deg; joints [-11.919, -28.167, 111.597, -15.944, -82.818, 51.029]
  Set speed (30.0 mm/s)
  Call Extruder(0.140)
  MoveL 9348 to (504.2, 495.8, 17.9) mm, rotated rx 0 ry 90 rz 0 deg; joints [-11.544, -28.115, 111.275, -15.576, -82.546, 51.061]
  Set speed (120.0 mm/s)
  MoveL 9349 to (504.39, 495.61, 17.9) mm, rotated rx 0 ry 90 rz 0 deg; joints [-11.523, -28.112, 111.256, -15.556, -82.531, 51.063]
  Set speed (30.0 mm/s)
  Call Extruder(0.203)
  MoveL 9350 to (509.32, 490.68, 17.9) mm, rotated rx 0 ry 90 rz 0 deg; joints [-10.985, -28.034, 110.781, -15.027, -82.13, 51.104]
  MoveL 9351 to (509.44, 490.56, 17.9) mm, rotated rx 0 ry 90 rz 0 deg; joints [-10.972, -28.032, 110.769, -15.014, -82.12, 51.105]
  Set speed (120.0 mm/s)
  MoveL 9352 to (490.47, 509.53, 17.9) mm, rotated rx 0 ry 90 rz 0 deg; joints [-13.08, -28.315, 112.553, -17.086, -83.628, 50.918]
  Set speed (1000.0 mm/s)
  MoveL 9353 to (490.4, 509.6, 17.9) mm, rotated rx 0 ry 90 rz 0 deg; joints [-13.088, -28.316, 112.559, -17.094, -83.634, 50.918]
  Set speed (15.0 mm/s)
  Call Extruder(0.559)
  MoveL 9354 to (490.4, 490.4, 17.9) mm, rotated rx 0 ry 90 rz 0 deg; joints [-11.303, -28.388, 113.05, -15.286, -83.988, 50.634]
  MoveL 9355 to (509.6, 490.4, 17.9) mm, rotated rx 0 ry 90 rz 0 deg; joints [-10.955, -28.029, 110.754, -14.998, -82.107, 51.106]
  MoveL 9356 to (509.6, 509.6, 17.9) mm, rotated rx 0 ry 90 rz 0 deg; joints [-12.688, -27.946, 110.268, -16.762, -81.782, 51.437]
  MoveL 9357 to (490.4, 509.6, 17.9) mm, rotated rx 0 ry 90 rz 0 deg; joints [-13.088, -28.316, 112.559, -17.094, -83.634, 50.918]
  Set speed (120.0 mm/s)
  MoveL 9358 to (490.4, 509.2, 17.9) mm, rotated rx 0 ry 90 rz 0 deg; joints [-13.051, -28.317, 112.57, -17.056, -83.642, 50.911]
  Set speed (1000.0 mm/s)
  MoveL 9359 to (490.5, 509.2, 17.9) mm, rotated rx 0 ry 90 rz 0 deg; joints [-13.049, -28.316, 112.558, -17.054, -83.632, 50.914]
  Set speed (1000.0 mm/s)
  MoveL 9360 to (496.05, 506.68, 17.9) mm, rotated rx 0 ry 90 rz 0 deg; joints [-12.7, -28.226, 111.97, -16.72, -83.144, 51.025]
  Set speed (15.0 mm/s)
  Call Extruder(0.065)
  MoveL 9361 to (496.05, 504.45, 17.9) mm, rotated rx 0 ry 90 rz 0 deg; joints [-12.495, -28.235, 112.029, -16.512, -83.185, 50.989]
  Call Extruder(0.145)
  MoveL 9362 to (501.03, 504.45, 17.9) mm, rotated rx 0 ry 90 rz 0 deg; joints [-12.394, -28.141, 111.435, -16.428, -82.703, 51.121]
  Call Extruder(0.353)
  MoveL 9363 to (495.52, 493.65, 17.9) mm, rotated rx 0 ry 90 rz 0 deg; joints [-11.509, -28.287, 112.365, -15.511, -83.43, 50.809]
  Call Extruder(0.261)
  MoveL 9364 to (504.47, 493.65, 17.9) mm, rotated rx 0 ry 90 rz 0 deg; joints [-11.343, -28.118, 111.294, -15.373, -82.555, 51.033]
  Call Extruder(0.065)
  MoveL 9365 to (504.47, 495.88, 17.9) mm, rotated rx 0 ry 90 rz 0 deg; joints [-11.547, -28.11, 111.24, -15.58, -82.518, 51.069]
  Call Extruder(0.153)
  MoveL 9366 to (499.2, 495.88, 17.9) mm, rotated rx 0 ry 90 rz 0 deg; joints [-11.646, -28.211, 111.871, -15.661, -83.031, 50.936]
  Call Extruder(0.353)
  MoveL 9367 to (504.73, 506.68, 17.9) mm, rotated rx 0 ry 90 rz 0 deg; joints [-12.523, -28.059, 110.933, -16.574, -82.304, 51.256]
  Call Extruder(0.253)
  MoveL 9368 to (496.05, 506.68, 17.9) mm, rotated rx 0 ry 90 rz 0 deg; joints [-12.7, -28.226, 111.97, -16.72, -83.144, 51.025]
  Set speed (120.0 mm/s)
  MoveL 9369 to (496.46, 506.36, 17.9) mm, rotated rx 0 ry 90 rz 0 deg; joints [-12.662, -28.22, 111.929, -16.683, -83.109, 51.031]
  Set speed (15.0 mm/s)
  Call Extruder(0.004)
  MoveL 9370 to (496.36, 506.26, 17.9) mm, rotated rx 0 ry 90 rz 0 deg; joints [-12.655, -28.222, 111.943, -16.676, -83.121, 51.027]
  Set speed (120.0 mm/s)
  MoveL 9371 to (496.36, 505.27, 17.9) mm, rotated rx 0 ry 90 rz 0 deg; joints [-12.564, -28.226, 111.97, -16.584, -83.14, 51.011]
  Set speed (15.0 mm/s)
  Call Extruder(0.045)
  MoveL 9372 to (497.45, 506.36, 17.9) mm, rotated rx 0 ry 90 rz 0 deg; joints [-12.642, -28.201, 111.811, -16.666, -83.014, 51.057]
  Set speed (120.0 mm/s)
  MoveL 9373 to (498.44, 506.36, 17.9) mm, rotated rx 0 ry 90 rz 0 deg; joints [-12.622, -28.183, 111.693, -16.65, -82.918, 51.084]
  Set speed (15.0 mm/s)
  Call Extruder(0.066)
  MoveL 9374 to (496.84, 504.76, 17.9) mm, rotated rx 0 ry 90 rz 0 deg; joints [-12.508, -28.219, 111.926, -16.528, -83.103, 51.015]
  Set speed (120.0 mm/s)
  MoveL 9375 to (497.83, 504.76, 17.9) mm, rotated rx 0 ry 90 rz 0 deg; joints [-12.488, -28.201, 111.809, -16.511, -83.007, 51.041]
  Set speed (15.0 mm/s)
  MoveL 9376 to (499.43, 506.36, 17.9) mm, rotated rx 0 ry 90 rz 0 deg; joints [-12.602, -28.164, 111.575, -16.633, -82.822, 51.11]
  Set speed (120.0 mm/s)
  MoveL 9377 to (500.42, 506.36, 17.9) mm, rotated rx 0 ry 90 rz 0 deg; joints [-12.581, -28.145, 111.457, -16.616, -82.726, 51.137]
  Set speed (15.0 mm/s)
  MoveL 9378 to (498.82, 504.76, 17.9) mm, rotated rx 0 ry 90 rz 0 deg; joints [-12.468, -28.182, 111.691, -16.494, -82.911, 51.068]
  Set speed (120.0 mm/s)
  MoveL 9379 to (499.81, 504.76, 17.9) mm, rotated rx 0 ry 90 rz 0 deg; joints [-12.448, -28.163, 111.572, -16.478, -82.815, 51.094]
  Set speed (15.0 mm/s)
  MoveL 9380 to (501.41, 506.36, 17.9) mm, rotated rx 0 ry 90 rz 0 deg; joints [-12.561, -28.126, 111.338, -16.599, -82.631, 51.163]
  Set speed (120.0 mm/s)
  MoveL 9381 to (502.4, 506.36, 17.9) mm, rotated rx 0 ry 90 rz 0 deg; joints [-12.541, -28.106, 111.22, -16.583, -82.535, 51.189]
  Set speed (15.0 mm/s)
  MoveL 9382 to (500.8, 504.76, 17.9) mm, rotated rx 0 ry 90 rz 0 deg; joints [-12.428, -28.144, 111.454, -16.461, -82.719, 51.12]
  Set speed (120.0 mm/s)
  MoveL 9383 to (501.28, 504.25, 17.9) mm, rotated rx 0 ry 90 rz 0 deg; joints [-12.372, -28.137, 111.41, -16.406, -82.682, 51.124]
  Set speed (15.0 mm/s)
  Call Extruder(0.087)
  MoveL 9384 to (503.39, 506.36, 17.9) mm, rotated rx 0 ry 90 rz 0 deg; joints [-12.521, -28.087, 111.102, -16.566, -82.439, 51.215]
  Set speed (120.0 mm/s)
  MoveL 9385 to (504.04, 506.02, 17.9) mm, rotated rx 0 ry 90 rz 0 deg; joints [-12.477, -28.076, 111.033, -16.524, -82.383, 51.227]
  Set speed (15.0 mm/s)
  Call Extruder(0.156)
  MoveL 9386 to (500.25, 502.23, 17.9) mm, rotated rx 0 ry 90 rz 0 deg; joints [-12.208, -28.165, 111.585, -16.236, -82.818, 51.064]
  MoveL 9387 to (500.13, 502.11, 17.9) mm, rotated rx 0 ry 90 rz 0 deg; joints [-12.199, -28.168, 111.603, -16.226, -82.832, 51.059]
  Set speed (120.0 mm/s)
  MoveL 9388 to (501.96, 501.96, 17.9) mm, rotated rx 0 ry 90 rz 0 deg; joints [-12.15, -28.134, 111.388, -16.183, -82.657, 51.104]
  Set speed (15.0 mm/s)
  Call Extruder(0.155)
  MoveL 9389 to (498.19, 498.19, 17.9) mm, rotated rx 0 ry 90 rz 0 deg; joints [-11.878, -28.22, 111.934, -15.893, -83.09, 50.946]
  MoveL 9390 to (498.07, 498.07, 17.9) mm, rotated rx 0 ry 90 rz 0 deg; joints [-11.869, -28.223, 111.952, -15.884, -83.104, 50.941]
  Set speed (120.0 mm/s)
  MoveL 9391 to (499.89, 497.91, 17.9) mm, rotated rx 0 ry 90 rz 0 deg; joints [-11.819, -28.19, 111.739, -15.84, -82.93, 50.986]
  Set speed (15.0 mm/s)
  Call Extruder(0.155)
  MoveL 9392 to (496.13, 494.15, 17.9) mm, rotated rx 0 ry 90 rz 0 deg; joints [-11.544, -28.274, 112.28, -15.548, -83.362, 50.832]
  Set speed (120.0 mm/s)
  MoveL 9393 to (496.93, 493.96, 17.9) mm, rotated rx 0 ry 90 rz 0 deg; joints [-11.512, -28.26, 112.189, -15.518, -83.286, 50.85]
  Set speed (15.0 mm/s)
  Call Extruder(0.079)
  MoveL 9394 to (498.85, 495.88, 17.9) mm, rotated rx 0 ry 90 rz 0 deg; joints [-11.652, -28.217, 111.913, -15.667, -83.066, 50.927]
  Set speed (120.0 mm/s)
  MoveL 9395 to (499.52, 495.57, 17.9) mm, rotated rx 0 ry 90 rz 0 deg; joints [-11.611, -28.206, 111.84, -15.627, -83.006, 50.94]
  Set speed (15.0 mm/s)
  Call Extruder(0.066)
  MoveL 9396 to (497.92, 493.96, 17.9) mm, rotated rx 0 ry 90 rz 0 deg; joints [-11.493, -28.242, 112.071, -15.502, -83.19, 50.875]
  Set speed (120.0 mm/s)
  MoveL 9397 to (498.91, 493.96, 17.9) mm, rotated rx 0 ry 90 rz 0 deg; joints [-11.475, -28.223, 111.953, -15.487, -83.093, 50.899]
  Set speed (15.0 mm/s)
  MoveL 9398 to (500.51, 495.56, 17.9) mm, rotated rx 0 ry 90 rz 0 deg; joints [-11.592, -28.187, 111.722, -15.612, -82.909, 50.965]
  Set speed (120.0 mm/s)
  MoveL 9399 to (501.5, 495.57, 17.9) mm, rotated rx 0 ry 90 rz 0 deg; joints [-11.573, -28.168, 111.604, -15.596, -82.813, 50.99]
  Set speed (15.0 mm/s)
  MoveL 9400 to (499.9, 493.96, 17.9) mm, rotated rx 0 ry 90 rz 0 deg; joints [-11.456, -28.205, 111.834, -15.472, -82.996, 50.924]
  Set speed (120.0 mm/s)
  MoveL 9401 to (500.89, 493.96, 17.9) mm, rotated rx 0 ry 90 rz 0 deg; joints [-11.438, -28.186, 111.716, -15.456, -82.9, 50.949]
  Set speed (15.0 mm/s)
  MoveL 9402 to (502.49, 495.56, 17.9) mm, rotated rx 0 ry 90 rz 0 deg; joints [-11.555, -28.149, 111.485, -15.581, -82.716, 51.014]
  Set speed (120.0 mm/s)
  MoveL 9403 to (503.48, 495.56, 17.9) mm, rotated rx 0 ry 90 rz 0 deg; joints [-11.536, -28.13, 111.366, -15.566, -82.62, 51.039]
  Set speed (15.0 mm/s)
  MoveL 9404 to (501.88, 493.96, 17.9) mm, rotated rx 0 ry 90 rz 0 deg; joints [-11.419, -28.167, 111.597, -15.441, -82.803, 50.974]
  Set speed (120.0 mm/s)
  MoveL 9405 to (502.87, 493.96, 17.9) mm, rotated rx 0 ry 90 rz 0 deg; joints [-11.401, -28.148, 111.479, -15.426, -82.706, 50.999]
  Set speed (15.0 mm/s)
  Call Extruder(0.053)
  MoveL 9406 to (504.16, 495.25, 17.9) mm, rotated rx 0 ry 90 rz 0 deg; joints [-11.495, -28.118, 111.293, -15.526, -82.559, 51.051]
  Set speed (120.0 mm/s)
  MoveL 9407 to (504.16, 494.26, 17.9) mm, rotated rx 0 ry 90 rz 0 deg; joints [-11.404, -28.122, 111.317, -15.434, -82.576, 51.035]
  Set speed (15.0 mm/s)
  Call Extruder(0.012)
  MoveL 9408 to (503.86, 493.96, 17.9) mm, rotated rx 0 ry 90 rz 0 deg; joints [-11.383, -28.129, 111.36, -15.411, -82.61, 51.023]
  Set speed (120.0 mm/s)
  MoveL 9409 to (500.93, 499.94, 17.9) mm, rotated rx 0 ry 90 rz 0 deg; joints [-11.985, -28.162, 111.564, -16.012, -82.793, 51.045]
  Set speed (15.0 mm/s)
  Call Extruder(0.155)
  MoveL 9410 to (497.16, 496.17, 17.9) mm, rotated rx 0 ry 90 rz 0 deg; joints [-11.711, -28.247, 112.108, -15.721, -83.226, 50.889]
  MoveL 9411 to (497.04, 496.05, 17.9) mm, rotated rx 0 ry 90 rz 0 deg; joints [-11.702, -28.25, 112.125, -15.711, -83.24, 50.884]
  Set speed (120.0 mm/s)
  MoveL 9412 to (499.22, 500.21, 17.9) mm, rotated rx 0 ry 90 rz 0 deg; joints [-12.043, -28.193, 111.76, -16.065, -82.954, 51.005]
  Set speed (15.0 mm/s)
  Call Extruder(0.156)
  MoveL 9413 to (503, 503.99, 17.9) mm, rotated rx 0 ry 90 rz 0 deg; joints [-12.314, -28.105, 111.211, -16.354, -82.52, 51.165]
  MoveL 9414 to (503.12, 504.12, 17.9) mm, rotated rx 0 ry 90 rz 0 deg; joints [-12.323, -28.102, 111.193, -16.363, -82.506, 51.17]
  Set speed (120.0 mm/s)
  MoveL 9415 to (490.68, 490.68, 17.9) mm, rotated rx 0 ry 90 rz 0 deg; joints [-11.324, -28.382, 113.01, -15.308, -83.956, 50.644]
  Set speed (1000.0 mm/s)
  MoveL 9416 to (490.68, 490.68, 18) mm, rotated rx 0 ry 90 rz 0 deg; joints [-11.324, -28.393, 113.016, -15.308, -83.95, 50.646]
  Set speed (30.0 mm/s)
  Call Extruder(0.287)
  MoveL 9417 to (497.65, 497.65, 18) mm, rotated rx 0 ry 90 rz 0 deg; joints [-11.838, -28.243, 112.017, -15.852, -83.147, 50.926]
  MoveL 9418 to (497.78, 497.78, 18) mm, rotated rx 0 ry 90 rz 0 deg; joints [-11.847, -28.24, 111.999, -15.861, -83.132, 50.931]
  Set speed (120.0 mm/s)
  MoveL 9419 to (499.24, 500.76, 18) mm, rotated rx 0 ry 90 rz 0 deg; joints [-12.093, -28.201, 111.75, -16.116, -82.937, 51.016]
  Set speed (30.0 mm/s)
  Call Extruder(0.352)
  MoveL 9420 to (490.68, 509.32, 18) mm, rotated rx 0 ry 90 rz 0 deg; joints [-13.056, -28.323, 112.539, -17.062, -83.607, 50.923]
  MoveL 9421 to (490.56, 509.44, 18) mm, rotated rx 0 ry 90 rz 0 deg; joints [-13.07, -28.324, 112.55, -17.076, -83.616, 50.921]
  Set speed (120.0 mm/s)
  MoveL 9422 to (496.13, 506.03, 18) mm, rotated rx 0 ry 90 rz 0 deg; joints [-12.639, -28.238, 111.983, -16.658, -83.143, 51.018]
  Set speed (30.0 mm/s)
  Call Extruder(0.224)
  MoveL 9423 to (490.68, 500.58, 18) mm, rotated rx 0 ry 90 rz 0 deg; joints [-12.247, -28.357, 112.771, -16.242, -83.773, 50.788]
  Set speed (120.0 mm/s)
  MoveL 9424 to (490.68, 499.42, 18) mm, rotated rx 0 ry 90 rz 0 deg; joints [-12.139, -28.361, 112.801, -16.133, -83.795, 50.771]
  Set speed (30.0 mm/s)
  Call Extruder(0.215)
  MoveL 9425 to (495.89, 494.2, 18) mm, rotated rx 0 ry 90 rz 0 deg; joints [-11.554, -28.288, 112.312, -15.557, -83.378, 50.828]
  Set speed (120.0 mm/s)
  MoveL 9426 to (496.37, 493.73, 18) mm, rotated rx 0 ry 90 rz 0 deg; joints [-11.5, -28.281, 112.266, -15.505, -83.34, 50.833]
  Set speed (30.0 mm/s)
  Call Extruder(0.125)
  MoveL 9427 to (499.42, 490.68, 18) mm, rotated rx 0 ry 90 rz 0 deg; joints [-11.163, -28.237, 111.976, -15.173, -83.093, 50.864]
  Set speed (120.0 mm/s)
  MoveL 9428 to (500.58, 490.68, 18) mm, rotated rx 0 ry 90 rz 0 deg; joints [-11.141, -28.215, 111.837, -15.155, -82.98, 50.892]
  Set speed (30.0 mm/s)
  MoveL 9429 to (503.63, 493.73, 18) mm, rotated rx 0 ry 90 rz 0 deg; joints [-11.366, -28.145, 111.399, -15.393, -82.631, 51.015]
  Set speed (120.0 mm/s)
  MoveL 9430 to (504.39, 494.49, 18) mm, rotated rx 0 ry 90 rz 0 deg; joints [-11.421, -28.127, 111.289, -15.452, -82.544, 51.046]
  Set speed (30.0 mm/s)
  Call Extruder(0.203)
  MoveL 9431 to (509.32, 499.42, 18) mm, rotated rx 0 ry 90 rz 0 deg; joints [-11.777, -28.008, 110.574, -15.833, -81.982, 51.251]
  Set speed (120.0 mm/s)
  MoveL 9432 to (509.32, 500.58, 18) mm, rotated rx 0 ry 90 rz 0 deg; joints [-11.882, -28.003, 110.544, -15.94, -81.962, 51.271]
  Set speed (30.0 mm/s)
  Call Extruder(0.212)
  MoveL 9433 to (504.16, 505.74, 18) mm, rotated rx 0 ry 90 rz 0 deg; joints [-12.449, -28.085, 111.031, -16.496, -82.371, 51.227]
  Set speed (120.0 mm/s)
  MoveL 9434 to (503.3, 506.6, 18) mm, rotated rx 0 ry 90 rz 0 deg; joints [-12.544, -28.098, 111.111, -16.59, -82.439, 51.219]
  Set speed (30.0 mm/s)
  Call Extruder(0.112)
  MoveL 9435 to (500.58, 509.32, 18) mm, rotated rx 0 ry 90 rz 0 deg; joints [-12.847, -28.139, 111.363, -16.887, -82.651, 51.192]
  Set speed (120.0 mm/s)
  MoveL 9436 to (499.42, 509.32, 18) mm, rotated rx 0 ry 90 rz 0 deg; joints [-12.872, -28.162, 111.502, -16.907, -82.763, 51.161]
  Set speed (30.0 mm/s)
  Call Extruder(0.112)
  MoveL 9437 to (496.7, 506.6, 18) mm, rotated rx 0 ry 90 rz 0 deg; joints [-12.679, -28.225, 111.899, -16.702, -83.077, 51.043]
  MoveL 9438 to (496.57, 506.47, 18) mm, rotated rx 0 ry 90 rz 0 deg; joints [-12.67, -28.228, 111.917, -16.692, -83.091, 51.037]
  Set speed (120.0 mm/s)
  MoveL 9439 to (502.51, 502.51, 18) mm, rotated rx 0 ry 90 rz 0 deg; joints [-12.188, -28.131, 111.314, -16.225, -82.589, 51.129]
  Set speed (30.0 mm/s)
  Call Extruder(0.280)
  MoveL 9440 to (509.32, 509.32, 18) mm, rotated rx 0 ry 90 rz 0 deg; joints [-12.669, -27.964, 110.315, -16.741, -81.809, 51.426]
  MoveL 9441 to (509.44, 509.44, 18) mm, rotated rx 0 ry 90 rz 0 deg; joints [-12.677, -27.961, 110.297, -16.751, -81.795, 51.431]
  Set speed (120.0 mm/s)
  MoveL 9442 to (500.81, 499.19, 18) mm, rotated rx 0 ry 90 rz 0 deg; joints [-11.919, -28.178, 111.602, -15.944, -82.812, 51.031]
  Set speed (30.0 mm/s)
  Call Extruder(0.140)
  MoveL 9443 to (504.2, 495.8, 18) mm, rotated rx 0 ry 90 rz 0 deg; joints [-11.544, -28.126, 111.28, -15.577, -82.541, 51.062]
  Set speed (120.0 mm/s)
  MoveL 9444 to (504.39, 495.61, 18) mm, rotated rx 0 ry 90 rz 0 deg; joints [-11.523, -28.123, 111.261, -15.556, -82.525, 51.064]
  Set speed (30.0 mm/s)
  Call Extruder(0.203)
  MoveL 9445 to (509.32, 490.68, 18) mm, rotated rx 0 ry 90 rz 0 deg; joints [-10.985, -28.044, 110.786, -15.027, -82.125, 51.105]
  MoveL 9446 to (509.44, 490.56, 18) mm, rotated rx 0 ry 90 rz 0 deg; joints [-10.972, -28.042, 110.774, -15.014, -82.115, 51.106]
  Set speed (120.0 mm/s)
  MoveL 9447 to (490.47, 509.53, 18) mm, rotated rx 0 ry 90 rz 0 deg; joints [-13.08, -28.326, 112.558, -17.086, -83.623, 50.92]
  Set speed (1000.0 mm/s)
  MoveL 9448 to (490.4, 509.6, 18) mm, rotated rx 0 ry 90 rz 0 deg; joints [-13.088, -28.326, 112.564, -17.094, -83.628, 50.919]
  Set speed (15.0 mm/s)
  Call Extruder(0.559)
  MoveL 9449 to (490.4, 490.4, 18) mm, rotated rx 0 ry 90 rz 0 deg; joints [-11.303, -28.398, 113.055, -15.287, -83.982, 50.635]
  MoveL 9450 to (509.6, 490.4, 18) mm, rotated rx 0 ry 90 rz 0 deg; joints [-10.955, -28.04, 110.759, -14.998, -82.102, 51.108]
  MoveL 9451 to (509.6, 509.6, 18) mm, rotated rx 0 ry 90 rz 0 deg; joints [-12.688, -27.957, 110.273, -16.763, -81.777, 51.438]
  MoveL 9452 to (490.4, 509.6, 18) mm, rotated rx 0 ry 90 rz 0 deg; joints [-13.088, -28.326, 112.564, -17.094, -83.628, 50.919]
  Set speed (120.0 mm/s)
  MoveL 9453 to (490.4, 509.2, 18) mm, rotated rx 0 ry 90 rz 0 deg; joints [-13.051, -28.328, 112.575, -17.056, -83.636, 50.913]
  Set speed (1000.0 mm/s)
  MoveL 9454 to (490.5, 509.2, 18) mm, rotated rx 0 ry 90 rz 0 deg; joints [-13.049, -28.326, 112.564, -17.054, -83.627, 50.916]
  Set speed (1000.0 mm/s)
  MoveL 9455 to (496.05, 506.68, 18) mm, rotated rx 0 ry 90 rz 0 deg; joints [-12.7, -28.237, 111.975, -16.72, -83.139, 51.026]
  Set speed (15.0 mm/s)
  Call Extruder(0.065)
  MoveL 9456 to (496.05, 504.45, 18) mm, rotated rx 0 ry 90 rz 0 deg; joints [-12.495, -28.246, 112.034, -16.512, -83.18, 50.991]
  Call Extruder(0.145)
  MoveL 9457 to (501.03, 504.45, 18) mm, rotated rx 0 ry 90 rz 0 deg; joints [-12.394, -28.152, 111.44, -16.429, -82.697, 51.122]
  Call Extruder(0.353)
  MoveL 9458 to (495.52, 493.65, 18) mm, rotated rx 0 ry 90 rz 0 deg; joints [-11.509, -28.297, 112.37, -15.511, -83.425, 50.811]
  Call Extruder(0.261)
  MoveL 9459 to (504.47, 493.65, 18) mm, rotated rx 0 ry 90 rz 0 deg; joints [-11.343, -28.129, 111.299, -15.373, -82.55, 51.035]
  Call Extruder(0.065)
  MoveL 9460 to (504.47, 495.88, 18) mm, rotated rx 0 ry 90 rz 0 deg; joints [-11.547, -28.12, 111.245, -15.58, -82.513, 51.071]
  Call Extruder(0.153)
  MoveL 9461 to (499.21, 495.88, 18) mm, rotated rx 0 ry 90 rz 0 deg; joints [-11.646, -28.221, 111.876, -15.662, -83.026, 50.938]
  Call Extruder(0.353)
  MoveL 9462 to (504.73, 506.68, 18) mm, rotated rx 0 ry 90 rz 0 deg; joints [-12.523, -28.069, 110.938, -16.574, -82.299, 51.258]
  Call Extruder(0.253)
  MoveL 9463 to (496.05, 506.68, 18) mm, rotated rx 0 ry 90 rz 0 deg; joints [-12.7, -28.237, 111.975, -16.72, -83.139, 51.026]
  Set speed (120.0 mm/s)
  MoveL 9464 to (503.93, 505.81, 18) mm, rotated rx 0 ry 90 rz 0 deg; joints [-12.461, -28.089, 111.056, -16.507, -82.392, 51.222]
  Set speed (15.0 mm/s)
  Call Extruder(0.023)
  MoveL 9465 to (503.39, 506.36, 18) mm, rotated rx 0 ry 90 rz 0 deg; joints [-12.521, -28.098, 111.107, -16.567, -82.435, 51.217]
  Set speed (120.0 mm/s)
  MoveL 9466 to (502.4, 506.36, 18) mm, rotated rx 0 ry 90 rz 0 deg; joints [-12.541, -28.117, 111.226, -16.583, -82.53, 51.191]
  Set speed (15.0 mm/s)
  Call Extruder(0.049)
  MoveL 9467 to (503.6, 505.16, 18) mm, rotated rx 0 ry 90 rz 0 deg; joints [-12.408, -28.099, 111.114, -16.452, -82.436, 51.202]
  Set speed (120.0 mm/s)
  MoveL 9468 to (503.26, 504.5, 18) mm, rotated rx 0 ry 90 rz 0 deg; joints [-12.355, -28.108, 111.171, -16.397, -82.48, 51.182]
  Set speed (15.0 mm/s)
  Call Extruder(0.076)
  MoveL 9469 to (501.41, 506.36, 18) mm, rotated rx 0 ry 90 rz 0 deg; joints [-12.561, -28.136, 111.344, -16.6, -82.626, 51.164]
  Set speed (120.0 mm/s)
  MoveL 9470 to (500.42, 506.36, 18) mm, rotated rx 0 ry 90 rz 0 deg; joints [-12.581, -28.155, 111.463, -16.616, -82.722, 51.138]
  Set speed (15.0 mm/s)
  Call Extruder(0.103)
  MoveL 9471 to (502.93, 503.85, 18) mm, rotated rx 0 ry 90 rz 0 deg; joints [-12.302, -28.117, 111.228, -16.342, -82.524, 51.162]
  Set speed (120.0 mm/s)
  MoveL 9472 to (502.59, 503.19, 18) mm, rotated rx 0 ry 90 rz 0 deg; joints [-12.249, -28.127, 111.286, -16.287, -82.568, 51.143]
  Set speed (15.0 mm/s)
  Call Extruder(0.050)
  MoveL 9473 to (501.37, 504.42, 18) mm, rotated rx 0 ry 90 rz 0 deg; joints [-12.385, -28.145, 111.4, -16.42, -82.665, 51.131]
  Set speed (120.0 mm/s)
  MoveL 9474 to (501.03, 504.76, 18) mm, rotated rx 0 ry 90 rz 0 deg; joints [-12.423, -28.15, 111.432, -16.458, -82.692, 51.128]
  Set speed (15.0 mm/s)
  Call Extruder(0.066)
  MoveL 9475 to (499.43, 506.36, 18) mm, rotated rx 0 ry 90 rz 0 deg; joints [-12.602, -28.174, 111.581, -16.633, -82.817, 51.112]
  Set speed (120.0 mm/s)
  MoveL 9476 to (498.44, 506.36, 18) mm, rotated rx 0 ry 90 rz 0 deg; joints [-12.622, -28.193, 111.699, -16.65, -82.913, 51.085]
  Set speed (15.0 mm/s)
  MoveL 9477 to (500.04, 504.76, 18) mm, rotated rx 0 ry 90 rz 0 deg; joints [-12.443, -28.169, 111.55, -16.474, -82.788, 51.102]
  Set speed (120.0 mm/s)
  MoveL 9478 to (499.05, 504.76, 18) mm, rotated rx 0 ry 90 rz 0 deg; joints [-12.463, -28.188, 111.668, -16.491, -82.883, 51.075]
  Set speed (15.0 mm/s)
  MoveL 9479 to (497.45, 506.36, 18) mm, rotated rx 0 ry 90 rz 0 deg; joints [-12.642, -28.212, 111.817, -16.667, -83.009, 51.059]
  Set speed (120.0 mm/s)
  MoveL 9480 to (496.46, 506.36, 18) mm, rotated rx 0 ry 90 rz 0 deg; joints [-12.663, -28.23, 111.934, -16.684, -83.105, 51.032]
  Set speed (15.0 mm/s)
  MoveL 9481 to (498.06, 504.76, 18) mm, rotated rx 0 ry 90 rz 0 deg; joints [-12.483, -28.207, 111.786, -16.507, -82.979, 51.049]
  Set speed (120.0 mm/s)
  MoveL 9482 to (497.07, 504.76, 18) mm, rotated rx 0 ry 90 rz 0 deg; joints [-12.503, -28.226, 111.904, -16.524, -83.075, 51.023]
  Set speed (15.0 mm/s)
  Call Extruder(0.029)
  MoveL 9483 to (496.36, 505.47, 18) mm, rotated rx 0 ry 90 rz 0 deg; joints [-12.583, -28.236, 111.97, -16.602, -83.131, 51.015]
  Set speed (120.0 mm/s)
  MoveL 9484 to (500.7, 503.11, 18) mm, rotated rx 0 ry 90 rz 0 deg; joints [-12.279, -28.164, 111.514, -16.31, -82.753, 51.092]
  Set speed (15.0 mm/s)
  Call Extruder(0.050)
  MoveL 9485 to (501.92, 501.88, 18) mm, rotated rx 0 ry 90 rz 0 deg; joints [-12.143, -28.145, 111.4, -16.177, -82.657, 51.104]
  Set speed (120.0 mm/s)
  MoveL 9486 to (501.59, 501.23, 18) mm, rotated rx 0 ry 90 rz 0 deg; joints [-12.09, -28.154, 111.457, -16.121, -82.701, 51.084]
  Set speed (15.0 mm/s)
  MoveL 9487 to (500.36, 502.45, 18) mm, rotated rx 0 ry 90 rz 0 deg; joints [-12.226, -28.173, 111.571, -16.255, -82.798, 51.072]
  Set speed (120.0 mm/s)
  MoveL 9488 to (500.03, 501.8, 18) mm, rotated rx 0 ry 90 rz 0 deg; joints [-12.172, -28.182, 111.628, -16.199, -82.842, 51.053]
  Set speed (15.0 mm/s)
  Call Extruder(0.050)
  MoveL 9489 to (501.25, 500.58, 18) mm, rotated rx 0 ry 90 rz 0 deg; joints [-12.037, -28.164, 111.513, -16.066, -82.745, 51.065]
  Set speed (120.0 mm/s)
  MoveL 9490 to (500.92, 499.92, 18) mm, rotated rx 0 ry 90 rz 0 deg; joints [-11.983, -28.173, 111.57, -16.011, -82.789, 51.046]
  Set speed (15.0 mm/s)
  Call Extruder(0.050)
  MoveL 9491 to (499.7, 501.14, 18) mm, rotated rx 0 ry 90 rz 0 deg; joints [-12.119, -28.191, 111.685, -16.144, -82.886, 51.034]
  Set speed (120.0 mm/s)
  MoveL 9492 to (499.36, 500.49, 18) mm, rotated rx 0 ry 90 rz 0 deg; joints [-12.066, -28.2, 111.742, -16.088, -82.93, 51.014]
  Set speed (15.0 mm/s)
  Call Extruder(0.050)
  MoveL 9493 to (500.58, 499.27, 18) mm, rotated rx 0 ry 90 rz 0 deg; joints [-11.93, -28.182, 111.627, -15.955, -82.833, 51.026]
  Set speed (120.0 mm/s)
  MoveL 9494 to (500.25, 498.61, 18) mm, rotated rx 0 ry 90 rz 0 deg; joints [-11.876, -28.191, 111.683, -15.9, -82.877, 51.007]
  Set speed (15.0 mm/s)
  MoveL 9495 to (499.03, 499.83, 18) mm, rotated rx 0 ry 90 rz 0 deg; joints [-12.012, -28.209, 111.798, -16.033, -82.974, 50.995]
  Set speed (120.0 mm/s)
  MoveL 9496 to (498.69, 499.17, 18) mm, rotated rx 0 ry 90 rz 0 deg; joints [-11.958, -28.218, 111.855, -15.977, -83.018, 50.976]
  Set speed (15.0 mm/s)
  Call Extruder(0.050)
  MoveL 9497 to (499.91, 497.96, 18) mm, rotated rx 0 ry 90 rz 0 deg; joints [-11.823, -28.2, 111.74, -15.844, -82.921, 50.988]
  Set speed (120.0 mm/s)
